KUKA KRL program: MyProgram_313().src

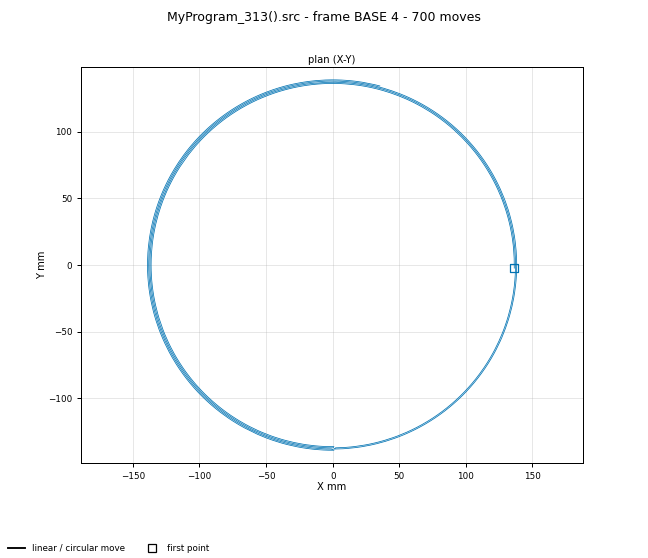
[picture p0: tool path of MyProgram_313().src in frame BASE 4, 700 of 700 moves have a stored position in this frame; points joined in program order, loops and branches not executed]
&ACCESS RVP
&REL 1
&PARAM TEMPLATE = C:\KRC\Roboter\Template\vorgabe
&PARAM EDITMASK = *
DEF MyProgram_313()
; ---- Setting reference (Base) ----
$BASE = BASE_DATA[4]

; --------------------------
; ---- Setting tool (TCP) ----
$TOOL = TOOL_DATA[3]
; --------------------------

$VEL.CP = VEL_APROX_PRINT
Startdeposition()
$VEL.CP = VEL_PRINT
LIN {X 136.3171,Y -2.3121,Z 183,A 1.901,B 4.2961,C 0.214,E1 4.4612,E2 450.9025} C_DIS
LIN {X 136.2426,Y 5.0697,Z 183,A 4.9757,B 4.2965,C 0.2056,E1 4.4611,E2 447.8295} C_DIS
LIN {X 135.7755,Y 12.3733,Z 183,A 8.1014,B 4.2969,C 0.1963,E1 4.4605,E2 444.6957} C_DIS
LIN {X 135.4586,Y 15.4613,Z 183,A 9.6734,B 4.2972,C 0.1892,E1 4.46,E2 443.0888} C_DIS
LIN {X 134.7828,Y 20.5264,Z 183,A 11.59,B 4.2974,C 0.1861,E1 4.4592,E2 441.2002} C_DIS
LIN {X 134.1353,Y 24.4028,Z 183,A 13.2335,B 4.2976,C 0.1816,E1 4.4584,E2 439.5567} C_DIS
LIN {X 133.2839,Y 28.6885,Z 183,A 14.8956,B 4.2976,C 0.1787,E1 4.4575,E2 437.9155} C_DIS
LIN {X 132.5463,Y 31.9229,Z 183,A 16.2711,B 4.2978,C 0.1751,E1 4.4566,E2 436.5415} C_DIS
LIN {X 131.506,Y 35.9772,Z 183,A 18.0412,B 4.298,C 0.1701,E1 4.4554,E2 434.7691} C_DIS
LIN {X 130.447,Y 39.6386,Z 183,A 19.5139,B 4.2981,C 0.1674,E1 4.4542,E2 433.3118} C_DIS
LIN {X 129.3994,Y 42.9345,Z 183,A 20.8992,B 4.2982,C 0.1643,E1 4.453,E2 431.9343} C_DIS
LIN {X 127.7702,Y 47.5649,Z 183,A 23.2775,B 4.2986,C 0.1549,E1 4.4507,E2 429.5151} C_DIS
LIN {X 126.4108,Y 51.0673,Z 183,A 24.4308,B 4.2986,C 0.156,E1 4.4496,E2 428.4147} C_DIS
LIN {X 125.0263,Y 54.3695,Z 183,A 25.8044,B 4.2986,C 0.1537,E1 4.4481,E2 427.0569} C_DIS
LIN {X 123.9979,Y 56.6781,Z 183,A 26.9937,B 4.2988,C 0.1494,E1 4.4467,E2 425.8511} C_DIS
LIN {X 122.4235,Y 60.0012,Z 183,A 28.472,B 4.2988,C 0.1462,E1 4.4449,E2 424.3805} C_DIS
LIN {X 120.7175,Y 63.3624,Z 183,A 29.8705,B 4.299,C 0.1445,E1 4.4431,E2 423.0045} C_DIS
LIN {X 118.9072,Y 66.7021,Z 183,A 31.598,B 4.2991,C 0.1389,E1 4.4408,E2 421.2601} C_DIS
LIN {X 116.1505,Y 71.3944,Z 183,A 33.7773,B 4.2993,C 0.1346,E1 4.4377,E2 419.0935} C_DIS
LIN {X 114.0434,Y 74.7147,Z 183,A 35.456,B 4.2994,C 0.1304,E1 4.4351,E2 417.411} C_DIS
LIN {X 111.5779,Y 78.3489,Z 183,A 37.2621,B 4.2995,C 0.1265,E1 4.4323,E2 415.6092} C_DIS
LIN {X 108.8614,Y 82.081,Z 183,A 38.9007,B 4.2995,C 0.1256,E1 4.4296,E2 414.0075} C_DIS
LIN {X 106.5784,Y 85.0244,Z 183,A 40.3825,B 4.2996,C 0.1231,E1 4.4271,E2 412.5356} C_DIS
LIN {X 103.9871,Y 88.1748,Z 183,A 42.3281,B 4.2998,C 0.1166,E1 4.4236,E2 410.5609} C_DIS
LIN {X 100.9585,Y 91.6267,Z 183,A 44.0964,B 4.2998,C 0.1144,E1 4.4203,E2 408.8123} C_DIS
LIN {X 96.8115,Y 95.9981,Z 183,A 46.6115,B 4.3,C 0.1093,E1 4.4155,E2 406.2989} C_DIS
LIN {X 91.1892,Y 101.3543,Z 183,A 49.8778,B 4.3002,C 0.1029,E1 4.4088,E2 403.0318} C_DIS
LIN {X 87.8086,Y 104.2966,Z 183,A 51.5269,B 4.3002,C 0.102,E1 4.4053,E2 401.4114} C_DIS
LIN {X 84.7834,Y 106.7702,Z 183,A 53.4489,B 4.3003,C 0.0958,E1 4.4011,E2 399.4547} C_DIS
LIN {X 80.5427,Y 110.0046,Z 183,A 55.502,B 4.3003,C 0.0941,E1 4.3965,E2 397.4248} C_DIS
LIN {X 76.9236,Y 112.5652,Z 183,A 57.3399,B 4.3004,C 0.0913,E1 4.3923,E2 395.5898} C_DIS
LIN {X 73.3431,Y 114.93,Z 183,A 59.0894,B 4.3004,C 0.089,E1 4.3882,E2 393.8469} C_DIS
LIN {X 69.468,Y 117.3134,Z 183,A 61.0062,B 4.3005,C 0.086,E1 4.3837,E2 391.9296} C_DIS
LIN {X 66.9374,Y 118.775,Z 183,A 62.2865,B 4.3005,C 0.0837,E1 4.3805,E2 390.6429} C_DIS
LIN {X 62.2571,Y 121.2921,Z 183,A 64.3036,B 4.3005,C 0.083,E1 4.3756,E2 388.6525} C_DIS
LIN {X 59.1852,Y 122.8204,Z 183,A 65.7141,B 4.3006,C 0.0814,E1 4.3721,E2 387.2459} C_DIS
LIN {X 55.8943,Y 124.352,Z 183,A 67.2309,B 4.3006,C 0.0796,E1 4.3682,E2 385.7304} C_DIS
LIN {X 52.4095,Y 125.8603,Z 183,A 68.781,B 4.3006,C 0.0782,E1 4.3643,E2 384.1861} C_DIS
LIN {X 49.7936,Y 126.9186,Z 183,A 69.9784,B 4.3006,C 0.0768,E1 4.3612,E2 382.9875} C_DIS
LIN {X 46.3245,Y 128.2248,Z 183,A 71.4966,B 4.3007,C 0.0756,E1 4.3572,E2 381.4743} C_DIS
LIN {X 43.3026,Y 129.2769,Z 183,A 72.8612,B 4.3007,C 0.0741,E1 4.3536,E2 380.1076} C_DIS
LIN {X 37.5599,Y 131.0627,Z 183,A 75.4609,B 4.3007,C 0.0711,E1 4.3466,E2 377.4997} C_DIS
LIN {X 33.8613,Y 132.0648,Z 183,A 76.9228,B 4.3007,C 0.0714,E1 4.3427,E2 376.0562} C_DIS
LIN {X 30.4313,Y 132.8967,Z 183,A 78.3894,B 4.3008,C 0.0705,E1 4.3387,E2 374.5921} C_DIS
LIN {X 27.0813,Y 133.6197,Z 183,A 79.8394,B 4.3008,C 0.0694,E1 4.3347,E2 373.1413} C_DIS
LIN {X 23.0702,Y 134.3719,Z 183,A 81.6264,B 4.3008,C 0.0678,E1 4.3298,E2 371.3461} C_DIS
LIN {X 19.4171,Y 134.9468,Z 183,A 83.0775,B 4.3008,C 0.068,E1 4.3258,E2 369.908} C_DIS
LIN {X 15.7292,Y 135.4268,Z 183,A 84.7916,B 4.3008,C 0.0659,E1 4.321,E2 368.1761} C_DIS
LIN {X 9.2863,Y 136.0215,Z 183,A 87.4726,B 4.3008,C 0.0654,E1 4.3136,E2 365.5008} C_DIS
LIN {X 6.3135,Y 136.1914,Z 183,A 89.0135,B 4.3009,C 0.0625,E1 4.3092,E2 363.925} C_DIS
LIN {X 2.4068,Y 136.3155,Z 183,A 90.1857,B 4.3009,C 0.0666,E1 4.3061,E2 362.811} C_DIS
LIN {X -4.4919,Y 136.2645,Z 183,A 93.2409,B 4.3009,C 0.0651,E1 4.2975,E2 359.7382} C_DIS
LIN {X -7.6288,Y 136.1251,Z 183,A 94.8342,B 4.3009,C 0.0628,E1 4.293,E2 358.1122} C_DIS
LIN {X -11.2331,Y 135.8732,Z 183,A 96.4152,B 4.3009,C 0.0624,E1 4.2885,E2 356.5241} C_DIS
LIN {X -15.4058,Y 135.4654,Z 183,A 97.8169,B 4.3009,C 0.0661,E1 4.2848,E2 355.1675} C_DIS
LIN {X -19.1221,Y 134.9889,Z 183,A 99.3275,B 4.3009,C 0.0671,E1 4.2806,E2 353.6654} C_DIS
LIN {X -22.8425,Y 134.4099,Z 183,A 100.9834,B 4.3009,C 0.0671,E1 4.276,E2 352.0014} C_DIS
LIN {X -26.9856,Y 133.6392,Z 183,A 102.6495,B 4.3009,C 0.0688,E1 4.2715,E2 350.3491} C_DIS
LIN {X -30.2949,Y 132.9279,Z 183,A 104.1186,B 4.3009,C 0.0692,E1 4.2674,E2 348.8751} C_DIS
LIN {X -33.6005,Y 132.131,Z 183,A 105.5284,B 4.3009,C 0.0703,E1 4.2636,E2 347.4684} C_DIS
LIN {X -36.8669,Y 131.2572,Z 183,A 107.3431,B 4.3009,C 0.0679,E1 4.2586,E2 345.6065} C_DIS
LIN {X -40.3293,Y 130.2356,Z 183,A 108.5381,B 4.3008,C 0.0718,E1 4.2555,E2 344.4519} C_DIS
LIN {X -44.2179,Y 128.9673,Z 183,A 110.2866,B 4.3008,C 0.073,E1 4.2509,E2 342.7009} C_DIS
LIN {X -47.9543,Y 127.6243,Z 183,A 112.7044,B 4.3008,C 0.0684,E1 4.2444,E2 340.1923} C_DIS
LIN {X -53.3534,Y 125.4656,Z 183,A 114.5344,B 4.3008,C 0.0759,E1 4.2398,E2 338.4394} C_DIS
LIN {X -56.6873,Y 123.9937,Z 183,A 115.9395,B 4.3007,C 0.0786,E1 4.2363,E2 337.0507} C_DIS
LIN {X -60.5692,Y 122.1433,Z 183,A 118.2237,B 4.3007,C 0.077,E1 4.2304,E2 334.7094} C_DIS
LIN {X -64.1356,Y 120.3106,Z 183,A 119.788,B 4.3007,C 0.0801,E1 4.2266,E2 333.1611} C_DIS
LIN {X -68.8121,Y 117.699,Z 183,A 121.7265,B 4.3005,C 0.0855,E1 4.222,E2 331.2625} C_DIS
LIN {X -72.0312,Y 115.7566,Z 183,A 123.5706,B 4.3005,C 0.0858,E1 4.2175,E2 329.3873} C_DIS
LIN {X -76.0435,Y 113.162,Z 183,A 125.5858,B 4.3005,C 0.0888,E1 4.2128,E2 327.3728} C_DIS
LIN {X -79.7494,Y 110.5813,Z 183,A 127.2851,B 4.3004,C 0.0933,E1 4.209,E2 325.6992} C_DIS
LIN {X -83.2352,Y 107.9819,Z 183,A 129.5008,B 4.3004,C 0.0935,E1 4.204,E2 323.4374} C_DIS
LIN {X -87.134,Y 104.8609,Z 183,A 131.4864,B 4.3003,C 0.098,E1 4.1997,E2 321.4673} C_DIS
LIN {X -90.591,Y 101.8896,Z 183,A 133.3086,B 4.3002,C 0.1021,E1 4.1959,E2 319.658} C_DIS
LIN {X -93.6569,Y 99.0781,Z 183,A 135.4627,B 4.3002,C 0.1026,E1 4.1914,E2 317.4555} C_DIS
LIN {X -96.0676,Y 96.7424,Z 183,A 136.6668,B 4.3001,C 0.1068,E1 4.189,E2 316.2779} C_DIS
LIN {X -99.1593,Y 93.5709,Z 183,A 138.5814,B 4.3,C 0.1102,E1 4.1853,E2 314.3582} C_DIS
LIN {X -103.3949,Y 88.8684,Z 183,A 141.4274,B 4.2999,C 0.1145,E1 4.18,E2 311.4916} C_DIS
LIN {X -108.2215,Y 82.9229,Z 183,A 144.6315,B 4.2997,C 0.1216,E1 4.1745,E2 308.2919} C_DIS
LIN {X -114.6392,Y 73.7974,Z 183,A 149.4868,B 4.2994,C 0.1314,E1 4.1668,E2 303.4203} C_DIS
LIN {X -117.1451,Y 69.7504,Z 183,A 151.5284,B 4.2992,C 0.136,E1 4.1638,E2 301.3752} C_DIS
LIN {X -119.4339,Y 65.7552,Z 183,A 153.5195,B 4.2991,C 0.1403,E1 4.161,E2 299.3788} C_DIS
LIN {X -121.3098,Y 62.2224,Z 183,A 155.1705,B 4.2989,C 0.1448,E1 4.1589,E2 297.7327} C_DIS
LIN {X -122.8831,Y 59.054,Z 183,A 156.4617,B 4.2988,C 0.1498,E1 4.1574,E2 296.467} C_DIS
LIN {X -124.4309,Y 55.7179,Z 183,A 158.7322,B 4.2988,C 0.1491,E1 4.1547,E2 294.1077} C_DIS
LIN {X -126.1198,Y 51.788,Z 183,A 160.2755,B 4.2986,C 0.1554,E1 4.153,E2 292.5978} C_DIS
LIN {X -127.6596,Y 47.8601,Z 183,A 161.7935,B 4.2983,C 0.1617,E1 4.1515,E2 291.1127} C_DIS
LIN {X -129.1595,Y 43.6552,Z 183,A 163.9661,B 4.2983,C 0.1649,E1 4.1495,E2 288.9049} C_DIS
LIN {X -131.0998,Y 37.4294,Z 183,A 166.8614,B 4.298,C 0.1713,E1 4.1472,E2 285.9926} C_DIS
LIN {X -132.0998,Y 33.7234,Z 183,A 168.3203,B 4.2978,C 0.1767,E1 4.1461,E2 284.5541} C_DIS
LIN {X -132.8008,Y 30.8514,Z 183,A 170.296,B 4.2978,C 0.1755,E1 4.1449,E2 282.4877} C_DIS
LIN {X -133.8259,Y 26.047,Z 183,A 171.8547,B 4.2974,C 0.1845,E1 4.144,E2 280.9941} C_DIS
LIN {X -134.4481,Y 22.6131,Z 183,A 173.3375,B 4.2973,C 0.1885,E1 4.1433,E2 279.5103} C_DIS
LIN {X -134.9784,Y 19.1958,Z 183,A 174.8432,B 4.2971,C 0.1922,E1 4.1427,E2 277.9992} C_DIS
LIN {X -135.4712,Y 15.3557,Z 183,A 176.5479,B 4.2969,C 0.1963,E1 4.1421,E2 276.2861} C_DIS
LIN {X -135.8304,Y 11.7403,Z 183,A 178.1035,B 4.2967,C 0.2004,E1 4.1417,E2 274.7279} C_DIS
LIN {X -136.0632,Y 8.6339,Z 183,A 179.5198,B 4.2966,C 0.2035,E1 4.1414,E2 273.2991} C_DIS
LIN {X -136.2696,Y 4.3069,Z 183,A -178.5717,B 4.2964,C 0.2081,E1 4.1412,E2 271.381} C_DIS
LIN {X -136.3402,Y 0.0169,Z 183,A -176.6762,B 4.2961,C 0.2126,E1 4.1412,E2 269.4752} C_DIS
LIN {X -136.2832,Y -3.8175,Z 183,A -175.1085,B 4.2959,C 0.2174,E1 4.1412,E2 267.914} C_DIS
LIN {X -136.1045,Y -7.9634,Z 183,A -173.3102,B 4.2957,C 0.222,E1 4.1415,E2 266.1101} C_DIS
LIN {X -135.852,Y -11.4845,Z 183,A -171.7908,B 4.2955,C 0.226,E1 4.1419,E2 264.5871} C_DIS
LIN {X -135.4498,Y -15.5365,Z 183,A -169.9324,B 4.2952,C 0.2298,E1 4.1424,E2 262.7113} C_DIS
LIN {X -134.9598,Y -19.3256,Z 183,A -168.3468,B 4.295,C 0.2345,E1 4.143,E2 261.1292} C_DIS
LIN {X -134.3387,Y -23.2663,Z 183,A -166.5398,B 4.2948,C 0.2383,E1 4.1439,E2 259.3068} C_DIS
LIN {X -133.6182,Y -27.0889,Z 183,A -164.9906,B 4.2945,C 0.2434,E1 4.1447,E2 257.7693} C_DIS
LIN {X -132.8825,Y -30.4937,Z 183,A -163.4974,B 4.2943,C 0.2472,E1 4.1456,E2 256.2733} C_DIS
LIN {X -131.3136,Y -36.6651,Z 183,A -160.6385,B 4.2939,C 0.2533,E1 4.1476,E2 253.3929} C_DIS
LIN {X -130.3246,Y -40.0388,Z 183,A -159.0904,B 4.2937,C 0.2568,E1 4.1489,E2 251.8366} C_DIS
LIN {X -127.4621,Y -48.3873,Z 183,A -155.2423,B 4.2932,C 0.2658,E1 4.1525,E2 247.9729} C_DIS
LIN {X -126.0166,Y -52.0351,Z 183,A -153.5708,B 4.2929,C 0.2699,E1 4.1542,E2 246.2993} C_DIS
LIN {X -124.6389,Y -55.253,Z 183,A -152.0835,B 4.2927,C 0.2736,E1 4.1559,E2 244.8106} C_DIS
LIN {X -123.2925,Y -58.197,Z 183,A -150.6015,B 4.2925,C 0.2762,E1 4.1576,E2 243.3138} C_DIS
LIN {X -121.615,Y -61.6229,Z 183,A -148.8042,B 4.2923,C 0.2789,E1 4.1599,E2 241.4922} C_DIS
LIN {X -119.1403,Y -66.2853,Z 183,A -146.405,B 4.2921,C 0.283,E1 4.1632,E2 239.0706} C_DIS
LIN {X -117.4157,Y -69.2945,Z 183,A -145.1492,B 4.2918,C 0.2879,E1 4.1649,E2 237.8414} C_DIS
LIN {X -115.0574,Y -73.1442,Z 183,A -143.1656,B 4.2915,C 0.2918,E1 4.1678,E2 235.8474} C_DIS
LIN {X -112.577,Y -76.9063,Z 183,A -141.2209,B 4.2912,C 0.2958,E1 4.1709,E2 233.8967} C_DIS
LIN {X -110.2635,Y -80.1879,Z 183,A -139.4641,B 4.291,C 0.2991,E1 4.1738,E2 232.1315} C_DIS
LIN {X -107.429,Y -83.9477,Z 183,A -137.4443,B 4.2907,C 0.3031,E1 4.1772,E2 230.107} C_DIS
LIN {X -104.6125,Y -87.4321,Z 183,A -135.5524,B 4.2904,C 0.307,E1 4.1806,E2 228.2145} C_DIS
LIN {X -102.418,Y -89.9933,Z 183,A -134.0693,B 4.2903,C 0.3095,E1 4.1833,E2 226.7231} C_DIS
LIN {X -98.7006,Y -94.0548,Z 183,A -131.7155,B 4.2899,C 0.3138,E1 4.1878,E2 224.3646} C_DIS
LIN {X -96.2337,Y -96.5774,Z 183,A -130.3834,B 4.2896,C 0.3178,E1 4.1904,E2 223.0524} C_DIS
LIN {X -93.7595,Y -98.9814,Z 183,A -128.7043,B 4.2896,C 0.3188,E1 4.1938,E2 221.3438} C_DIS
LIN {X -90.5069,Y -101.964,Z 183,A -126.8241,B 4.2893,C 0.3219,E1 4.1977,E2 219.4605} C_DIS
LIN {X -87.0847,Y -104.9017,Z 183,A -124.8812,B 4.2891,C 0.3248,E1 4.2019,E2 217.5117} C_DIS
LIN {X -83.4222,Y -107.837,Z 183,A -122.8734,B 4.2889,C 0.3278,E1 4.2063,E2 215.4994} C_DIS
LIN {X -79.771,Y -110.5656,Z 183,A -121.0017,B 4.2886,C 0.3312,E1 4.2105,E2 213.6335} C_DIS
LIN {X -76.2754,Y -113.0052,Z 183,A -119.1733,B 4.2884,C 0.3336,E1 4.2147,E2 211.8003} C_DIS
LIN {X -73.143,Y -115.0581,Z 183,A -117.4666,B 4.2884,C 0.3348,E1 4.2188,E2 210.0763} C_DIS
LIN {X -69.7634,Y -117.1373,Z 183,A -115.7098,B 4.2882,C 0.3363,E1 4.223,E2 208.3079} C_DIS
LIN {X -65.4726,Y -119.5888,Z 183,A -113.6904,B 4.288,C 0.3394,E1 4.2279,E2 206.2959} C_DIS
LIN {X -62.3781,Y -121.2305,Z 183,A -112.2243,B 4.2879,C 0.3412,E1 4.2316,E2 204.8304} C_DIS
LIN {X -59.177,Y -122.8243,Z 183,A -110.8983,B 4.2876,C 0.3444,E1 4.2348,E2 203.5273} C_DIS
LIN {X -56.3296,Y -124.1573,Z 183,A -109.3311,B 4.2876,C 0.3437,E1 4.2389,E2 201.9279} C_DIS
LIN {X -52.8989,Y -125.6559,Z 183,A -107.8264,B 4.2875,C 0.3459,E1 4.2427,E2 200.4319} C_DIS
LIN {X -49.409,Y -127.0681,Z 183,A -106.2591,B 4.2874,C 0.3475,E1 4.2468,E2 198.8662} C_DIS
LIN {X -46.4075,Y -128.1949,Z 183,A -104.9422,B 4.2872,C 0.3489,E1 4.2502,E2 197.553} C_DIS
LIN {X -43.471,Y -129.2208,Z 183,A -103.3323,B 4.2874,C 0.3472,E1 4.2546,E2 195.9033} C_DIS
LIN {X -38.5666,Y -130.768,Z 183,A -101.3944,B 4.2871,C 0.3507,E1 4.2597,E2 193.9941} C_DIS
LIN {X -35.4538,Y -131.6462,Z 183,A -100.0022,B 4.2871,C 0.3513,E1 4.2635,E2 192.5972} C_DIS
LIN {X -32.1264,Y -132.4973,Z 183,A -98.557,B 4.287,C 0.352,E1 4.2674,E2 191.1514} C_DIS
LIN {X -29.0028,Y -133.216,Z 183,A -97.186,B 4.287,C 0.3525,E1 4.2711,E2 189.7768} C_DIS
LIN {X -25.6001,Y -133.9114,Z 183,A -95.7519,B 4.2869,C 0.3533,E1 4.2751,E2 188.3456} C_DIS
LIN {X -22.6007,Y -134.4502,Z 183,A -94.5199,B 4.2868,C 0.3542,E1 4.2784,E2 187.1195} C_DIS
LIN {X -19.4079,Y -134.9481,Z 183,A -92.2688,B 4.2875,C 0.3461,E1 4.285,E2 184.7502} C_DIS
LIN {X -13.2742,Y -135.689,Z 183,A -90.5042,B 4.2868,C 0.3545,E1 4.2896,E2 183.0945} C_DIS
LIN {X -9.9023,Y -135.9765,Z 183,A -88.6028,B 4.2871,C 0.35,E1 4.2951,E2 181.1294} C_DIS
LIN {X -5.6395,Y -136.2204,Z 183,A -87.4752,B 4.2866,C 0.3565,E1 4.298,E2 180.0887} C_DIS
LIN {X 0.9463,Y -136.3293,Z 183,A -85.9047,B 4.2856,C 0.3681,E1 4.3021,E2 178.6724} C_DIS
Enddeposition()
LIN {X 0.9463,Y -136.3293,Z 183,A -85.9053,B 4.2856,C 0.3681,E1 4.3021,E2 178.6731} C_DIS
Startdeposition()
$VEL.CP = VEL_PRINT
LIN {X 0.2601,Y -137.2384,Z 183,A -85.4933,B 4.2391,C 0.3624,E1 4.2564,E2 178.217} C_DIS
LIN {X -3.5849,Y -137.1911,Z 183,A -86.9897,B 4.2391,C 0.3615,E1 4.2522,E2 179.6999} C_DIS
LIN {X -8.3049,Y -136.9862,Z 183,A -89.3069,B 4.2389,C 0.3648,E1 4.2456,E2 182.0629} C_DIS
LIN {X -11.9801,Y -136.7144,Z 183,A -90.5859,B 4.2391,C 0.3622,E1 4.2421,E2 183.3087} C_DIS
LIN {X -16.1912,Y -136.2791,Z 183,A -92.2802,B 4.2392,C 0.3612,E1 4.2375,E2 184.9941} C_DIS
LIN {X -19.279,Y -135.8767,Z 183,A -94.0043,B 4.2389,C 0.3648,E1 4.2325,E2 186.774} C_DIS
LIN {X -23.4354,Y -135.2238,Z 183,A -95.4492,B 4.2392,C 0.3613,E1 4.2287,E2 188.179} C_DIS
LIN {X -27.2424,Y -134.5064,Z 183,A -96.8991,B 4.2394,C 0.3591,E1 4.2247,E2 189.6075} C_DIS
LIN {X -29.9628,Y -133.928,Z 183,A -98.1591,B 4.2394,C 0.3595,E1 4.2213,E2 190.8808} C_DIS
LIN {X -33.7684,Y -133.018,Z 183,A -99.7549,B 4.2394,C 0.3583,E1 4.2169,E2 192.472} C_DIS
LIN {X -37.2233,Y -132.0931,Z 183,A -101.3123,B 4.2394,C 0.3579,E1 4.2127,E2 194.0382} C_DIS
LIN {X -40.8878,Y -131.007,Z 183,A -103.0788,B 4.2394,C 0.3583,E1 4.2079,E2 195.8275} C_DIS
LIN {X -44.5595,Y -129.8025,Z 183,A -104.3666,B 4.2398,C 0.3542,E1 4.2046,E2 197.0731} C_DIS
LIN {X -47.8395,Y -128.6295,Z 183,A -105.9965,B 4.2398,C 0.3545,E1 4.2003,E2 198.7263} C_DIS
LIN {X -51.2367,Y -127.314,Z 183,A -107.5208,B 4.2398,C 0.3532,E1 4.1963,E2 200.2512} C_DIS
LIN {X -54.5588,Y -125.9261,Z 183,A -109.0138,B 4.24,C 0.3516,E1 4.1925,E2 201.7431} C_DIS
LIN {X -57.4805,Y -124.6196,Z 183,A -110.3802,B 4.2401,C 0.3504,E1 4.189,E2 203.1137} C_DIS
LIN {X -60.5172,Y -123.1736,Z 183,A -111.8923,B 4.2401,C 0.3498,E1 4.1852,E2 204.6399} C_DIS
LIN {X -63.6638,Y -121.577,Z 183,A -113.298,B 4.2404,C 0.3475,E1 4.1817,E2 206.0369} C_DIS
LIN {X -67.4381,Y -119.5271,Z 183,A -115.1334,B 4.2405,C 0.3456,E1 4.1772,E2 207.8781} C_DIS
LIN {X -70.8525,Y -117.5353,Z 183,A -116.9033,B 4.2406,C 0.3443,E1 4.1729,E2 209.6635} C_DIS
LIN {X -74.5041,Y -115.2553,Z 183,A -118.7553,B 4.2408,C 0.3422,E1 4.1685,E2 211.5227} C_DIS
LIN {X -78.2554,Y -112.7418,Z 183,A -120.6384,B 4.241,C 0.3394,E1 4.1642,E2 213.4054} C_DIS
LIN {X -81.7759,Y -110.2149,Z 183,A -122.5092,B 4.2412,C 0.3371,E1 4.1599,E2 215.2841} C_DIS
LIN {X -85.3945,Y -107.4354,Z 183,A -124.3352,B 4.2415,C 0.3333,E1 4.1559,E2 217.0998} C_DIS
LIN {X -88.1603,Y -105.1776,Z 183,A -126.1692,B 4.2415,C 0.3333,E1 4.1519,E2 218.978} C_DIS
LIN {X -90.708,Y -102.9889,Z 183,A -127.3956,B 4.2418,C 0.3295,E1 4.1494,E2 220.1816} C_DIS
LIN {X -93.9609,Y -100.0301,Z 183,A -129.2727,B 4.242,C 0.3265,E1 4.1455,E2 222.0638} C_DIS
LIN {X -96.2069,Y -97.8716,Z 183,A -130.8148,B 4.242,C 0.3258,E1 4.1424,E2 223.6367} C_DIS
LIN {X -98.5717,Y -95.4892,Z 183,A -131.7436,B 4.2425,C 0.3196,E1 4.1407,E2 224.5043} C_DIS
LIN {X -103.5219,Y -90.099,Z 183,A -135.1526,B 4.2428,C 0.316,E1 4.1342,E2 227.9585} C_DIS
LIN {X -106.4573,Y -86.6113,Z 183,A -137.107,B 4.2431,C 0.3124,E1 4.1307,E2 229.919} C_DIS
LIN {X -109.4579,Y -82.7862,Z 183,A -139.5581,B 4.2431,C 0.3109,E1 4.1264,E2 232.4234} C_DIS
LIN {X -111.8993,Y -79.4564,Z 183,A -141.0153,B 4.2436,C 0.3052,E1 4.1241,E2 233.8461} C_DIS
LIN {X -114.5103,Y -75.644,Z 183,A -142.9558,B 4.2439,C 0.3008,E1 4.1211,E2 235.7873} C_DIS
LIN {X -116.8963,Y -71.9018,Z 183,A -144.8729,B 4.2442,C 0.2969,E1 4.1182,E2 237.712} C_DIS
LIN {X -119.3495,Y -67.7522,Z 183,A -146.9295,B 4.2445,C 0.2924,E1 4.1154,E2 239.7734} C_DIS
LIN {X -121.3088,Y -64.1746,Z 183,A -148.7116,B 4.2448,C 0.2887,E1 4.113,E2 241.5648} C_DIS
LIN {X -123.0576,Y -60.7523,Z 183,A -150.2133,B 4.2451,C 0.284,E1 4.1111,E2 243.0528} C_DIS
LIN {X -124.4866,Y -57.768,Z 183,A -151.7131,B 4.2453,C 0.2813,E1 4.1093,E2 244.5671} C_DIS
LIN {X -126.0422,Y -54.2902,Z 183,A -153.312,B 4.2455,C 0.2773,E1 4.1075,E2 246.1662} C_DIS
LIN {X -127.3248,Y -51.2098,Z 183,A -154.7888,B 4.2457,C 0.2742,E1 4.1059,E2 247.653} C_DIS
LIN {X -128.4892,Y -48.2141,Z 183,A -156.451,B 4.2458,C 0.2728,E1 4.1043,E2 249.3551} C_DIS
LIN {X -129.6279,Y -45.063,Z 183,A -157.6634,B 4.2461,C 0.2679,E1 4.1032,E2 250.5432} C_DIS
LIN {X -130.9576,Y -41.0455,Z 183,A -159.5558,B 4.2464,C 0.264,E1 4.1015,E2 252.4507} C_DIS
LIN {X -132.0714,Y -37.3007,Z 183,A -161.11,B 4.2467,C 0.2591,E1 4.1003,E2 253.9942} C_DIS
LIN {X -133.2683,Y -32.7729,Z 183,A -163.2089,B 4.2469,C 0.2547,E1 4.0989,E2 256.1102} C_DIS
LIN {X -134.101,Y -29.173,Z 183,A -164.7257,B 4.2472,C 0.2503,E1 4.0979,E2 257.6228} C_DIS
LIN {X -134.7767,Y -25.8722,Z 183,A -166.1765,B 4.2474,C 0.2466,E1 4.0971,E2 259.0783} C_DIS
LIN {X -135.4035,Y -22.3621,Z 183,A -167.7293,B 4.2476,C 0.2429,E1 4.0964,E2 260.6383} C_DIS
LIN {X -136.0284,Y -18.181,Z 183,A -169.5698,B 4.2479,C 0.2384,E1 4.0957,E2 262.4872} C_DIS
LIN {X -136.4568,Y -14.6181,Z 183,A -170.9903,B 4.2481,C 0.2337,E1 4.0952,E2 263.8969} C_DIS
LIN {X -136.7536,Y -11.5159,Z 183,A -172.396,B 4.2483,C 0.2307,E1 4.0949,E2 265.315} C_DIS
LIN {X -136.9966,Y -8.1356,Z 183,A -174.0188,B 4.2484,C 0.228,E1 4.0946,E2 266.9629} C_DIS
LIN {X -137.1858,Y -3.7744,Z 183,A -175.8124,B 4.2487,C 0.2227,E1 4.0944,E2 268.7516} C_DIS
LIN {X -137.2396,Y -0.3029,Z 183,A -177.4372,B 4.2489,C 0.2197,E1 4.0944,E2 270.3974} C_DIS
LIN {X -137.1862,Y 3.7592,Z 183,A -179.0703,B 4.2491,C 0.2145,E1 4.0944,E2 272.0214} C_DIS
LIN {X -137.0072,Y 7.9645,Z 183,A 179.0956,B 4.2494,C 0.21,E1 4.0947,E2 273.8638} C_DIS
LIN {X -136.7496,Y 11.5627,Z 183,A 177.5779,B 4.2496,C 0.2058,E1 4.095,E2 275.3819} C_DIS
LIN {X -136.368,Y 15.4439,Z 183,A 175.7995,B 4.2498,C 0.2021,E1 4.0956,E2 277.1778} C_DIS
LIN {X -135.8787,Y 19.2647,Z 183,A 174.1963,B 4.25,C 0.1976,E1 4.0962,E2 278.7791} C_DIS
LIN {X -135.2411,Y 23.3353,Z 183,A 172.3171,B 4.2501,C 0.1937,E1 4.097,E2 280.6768} C_DIS
LIN {X -134.5025,Y 27.2619,Z 183,A 170.6317,B 4.2503,C 0.1892,E1 4.0979,E2 282.363} C_DIS
LIN {X -133.5396,Y 31.6473,Z 183,A 168.6557,B 4.2505,C 0.1847,E1 4.0992,E2 284.3502} C_DIS
LIN {X -132.5441,Y 35.5839,Z 183,A 166.9366,B 4.2507,C 0.1802,E1 4.1004,E2 286.0709} C_DIS
LIN {X -131.6299,Y 38.8295,Z 183,A 165.4351,B 4.2509,C 0.1769,E1 4.1016,E2 287.5829} C_DIS
LIN {X -130.3284,Y 42.9967,Z 183,A 163.606,B 4.2511,C 0.172,E1 4.1031,E2 289.4113} C_DIS
LIN {X -128.9393,Y 46.9993,Z 183,A 161.7571,B 4.2512,C 0.1678,E1 4.1049,E2 291.2687} C_DIS
LIN {X -127.6226,Y 50.4694,Z 183,A 160.2723,B 4.2514,C 0.1633,E1 4.1063,E2 292.7443} C_DIS
LIN {X -124.1756,Y 58.4387,Z 183,A 156.4308,B 4.2517,C 0.1553,E1 4.1107,E2 296.6097} C_DIS
LIN {X -122.4671,Y 61.9351,Z 183,A 154.8796,B 4.2519,C 0.1507,E1 4.1126,E2 298.1504} C_DIS
LIN {X -120.7035,Y 65.3101,Z 183,A 153.1135,B 4.2519,C 0.1479,E1 4.115,E2 299.937} C_DIS
LIN {X -118.5431,Y 69.1542,Z 183,A 151.1725,B 4.2521,C 0.144,E1 4.1177,E2 301.8887} C_DIS
LIN {X -116.1965,Y 73.0276,Z 183,A 149.3029,B 4.2523,C 0.1394,E1 4.1204,E2 303.7542} C_DIS
LIN {X -112.8084,Y 78.1596,Z 183,A 146.6334,B 4.2524,C 0.134,E1 4.1246,E2 306.4341} C_DIS
LIN {X -110.3698,Y 81.5674,Z 183,A 144.8068,B 4.2525,C 0.1306,E1 4.1276,E2 308.2687} C_DIS
LIN {X -107.6211,Y 85.1612,Z 183,A 142.8691,B 4.2527,C 0.1267,E1 4.1309,E2 310.2108} C_DIS
LIN {X -105.2665,Y 88.0544,Z 183,A 141.1005,B 4.2527,C 0.1248,E1 4.1341,E2 312.0039} C_DIS
LIN {X -101.563,Y 92.3014,Z 183,A 138.8869,B 4.2529,C 0.1189,E1 4.1382,E2 314.1987} C_DIS
LIN {X -98.5484,Y 95.5133,Z 183,A 137.0517,B 4.2529,C 0.1152,E1 4.1417,E2 316.032} C_DIS
LIN {X -95.8654,Y 98.2064,Z 183,A 135.4977,B 4.2531,C 0.1118,E1 4.1448,E2 317.5807} C_DIS
LIN {X -93.7361,Y 100.2407,Z 183,A 134.0774,B 4.2531,C 0.1108,E1 4.1477,E2 319.0232} C_DIS
LIN {X -90.3316,Y 103.3189,Z 183,A 132.1482,B 4.2531,C 0.1073,E1 4.1517,E2 320.9525} C_DIS
LIN {X -87.1051,Y 106.0538,Z 183,A 130.3098,B 4.2533,C 0.1047,E1 4.1557,E2 322.7983} C_DIS
LIN {X -84.2489,Y 108.3363,Z 183,A 128.9662,B 4.2533,C 0.1008,E1 4.1586,E2 324.1185} C_DIS
LIN {X -81.3703,Y 110.5146,Z 183,A 127.2372,B 4.2533,C 0.0999,E1 4.1625,E2 325.8734} C_DIS
LIN {X -77.6878,Y 113.1335,Z 183,A 125.3605,B 4.2534,C 0.0969,E1 4.1668,E2 327.7475} C_DIS
LIN {X -74.1226,Y 115.5009,Z 183,A 123.5147,B 4.2534,C 0.0946,E1 4.1711,E2 329.5991} C_DIS
LIN {X -71.0384,Y 117.4229,Z 183,A 121.7051,B 4.2534,C 0.0946,E1 4.1756,E2 331.4429} C_DIS
LIN {X -67.9666,Y 119.2272,Z 183,A 120.4764,B 4.2536,C 0.0907,E1 4.1784,E2 332.6394} C_DIS
LIN {X -65.2687,Y 120.7257,Z 183,A 118.4359,B 4.2535,C 0.0947,E1 4.1837,E2 334.7696} C_DIS
LIN {X -60.0003,Y 123.4286,Z 183,A 116.5624,B 4.2537,C 0.0872,E1 4.1882,E2 336.5694} C_DIS
LIN {X -56.4517,Y 125.0897,Z 183,A 115.0754,B 4.2537,C 0.0842,E1 4.1919,E2 338.0373} C_DIS
LIN {X -53.1906,Y 126.5105,Z 183,A 113.2957,B 4.2537,C 0.0849,E1 4.1966,E2 339.8516} C_DIS
LIN {X -49.0237,Y 128.1846,Z 183,A 111.5771,B 4.2537,C 0.0819,E1 4.201,E2 341.5501} C_DIS
LIN {X -45.4743,Y 129.4853,Z 183,A 110.0136,B 4.2537,C 0.0803,E1 4.2051,E2 343.1108} C_DIS
LIN {X -41.9569,Y 130.6665,Z 183,A 108.5035,B 4.2538,C 0.0787,E1 4.2091,E2 344.6152} C_DIS
LIN {X -39.0993,Y 131.5509,Z 183,A 107.3572,B 4.2538,C 0.077,E1 4.2121,E2 345.7484} C_DIS
LIN {X -35.6948,Y 132.5145,Z 183,A 105.7334,B 4.2538,C 0.0772,E1 4.2166,E2 347.3891} C_DIS
LIN {X -32.4552,Y 133.3448,Z 183,A 104.4011,B 4.2538,C 0.0758,E1 4.2201,E2 348.7128} C_DIS
LIN {X -29.1429,Y 134.1075,Z 183,A 103.0262,B 4.2538,C 0.0746,E1 4.2239,E2 350.0815} C_DIS
LIN {X -26.5653,Y 134.6442,Z 183,A 101.7012,B 4.2538,C 0.076,E1 4.2276,E2 351.4333} C_DIS
LIN {X -23.1425,Y 135.2733,Z 183,A 100.2784,B 4.2538,C 0.0751,E1 4.2315,E2 352.8516} C_DIS
LIN {X -19.2564,Y 135.8799,Z 183,A 98.6936,B 4.2539,C 0.074,E1 4.2358,E2 354.4286} C_DIS
LIN {X -15.59,Y 136.3508,Z 183,A 97.2032,B 4.2539,C 0.0732,E1 4.24,E2 355.9119} C_DIS
LIN {X -5.2554,Y 137.137,Z 183,A 92.7993,B 4.2539,C 0.0733,E1 4.2523,E2 360.3231} C_DIS
LIN {X 2.0919,Y 137.2219,Z 183,A 89.9384,B 4.2539,C 0.0716,E1 4.2602,E2 363.1577} C_DIS
LIN {X 9.3172,Y 136.9227,Z 183,A 85.9601,B 4.2538,C 0.0811,E1 4.2716,E2 367.2506} C_DIS
LIN {X 15.2036,Y 136.3938,Z 183,A 83.8558,B 4.2538,C 0.0787,E1 4.2773,E2 369.3105} C_DIS
LIN {X 19.1599,Y 135.8937,Z 183,A 82.6308,B 4.2538,C 0.0752,E1 4.2806,E2 370.4817} C_DIS
LIN {X 22.5717,Y 135.3685,Z 183,A 81.2103,B 4.2538,C 0.0758,E1 4.2845,E2 371.8993} C_DIS
LIN {X 26.2511,Y 134.7043,Z 183,A 79.6483,B 4.2538,C 0.0767,E1 4.2888,E2 373.4609} C_DIS
LIN {X 30.1207,Y 133.8919,Z 183,A 77.9549,B 4.2538,C 0.0782,E1 4.2934,E2 375.1591} C_DIS
LIN {X 33.7685,Y 133.018,Z 183,A 76.4358,B 4.2538,C 0.0789,E1 4.2975,E2 376.672} C_DIS
LIN {X 37.1198,Y 132.122,Z 183,A 75.0255,B 4.2538,C 0.0797,E1 4.3013,E2 378.0774} C_DIS
LIN {X 40.6062,Y 131.0932,Z 183,A 73.4777,B 4.2538,C 0.0814,E1 4.3054,E2 379.6285} C_DIS
LIN {X 44.7566,Y 129.7341,Z 183,A 71.7204,B 4.2538,C 0.0825,E1 4.3101,E2 381.3775} C_DIS
LIN {X 48.1002,Y 128.5318,Z 183,A 70.3349,B 4.2538,C 0.083,E1 4.3137,E2 382.7508} C_DIS
LIN {X 50.9035,Y 127.4483,Z 183,A 69.0172,B 4.2537,C 0.085,E1 4.3171,E2 384.076} C_DIS
LIN {X 54.1583,Y 126.0993,Z 183,A 67.5527,B 4.2537,C 0.0867,E1 4.3209,E2 385.5395} C_DIS
LIN {X 56.8125,Y 124.9283,Z 183,A 66.2204,B 4.2537,C 0.0894,E1 4.3243,E2 386.8864} C_DIS
LIN {X 60.3939,Y 123.2344,Z 183,A 64.6928,B 4.2536,C 0.0902,E1 4.3281,E2 388.3984} C_DIS
LIN {X 63.3851,Y 121.7233,Z 183,A 63.3232,B 4.2536,C 0.0918,E1 4.3315,E2 389.7644} C_DIS
LIN {X 67.3168,Y 119.5953,Z 183,A 61.4515,B 4.2535,C 0.0945,E1 4.3361,E2 391.6367} C_DIS
LIN {X 71.1732,Y 117.3414,Z 183,A 59.6076,B 4.2535,C 0.0971,E1 4.3405,E2 393.478} C_DIS
LIN {X 74.9729,Y 114.951,Z 183,A 57.7763,B 4.2534,C 0.0996,E1 4.3448,E2 395.3041} C_DIS
LIN {X 78.6365,Y 112.4766,Z 183,A 55.9552,B 4.2534,C 0.1023,E1 4.349,E2 397.1222} C_DIS
LIN {X 82.3156,Y 109.8131,Z 183,A 54.124,B 4.2533,C 0.1049,E1 4.3531,E2 398.9456} C_DIS
LIN {X 85.1425,Y 107.636,Z 183,A 52.6724,B 4.2533,C 0.1071,E1 4.3563,E2 400.3926} C_DIS
LIN {X 88.4415,Y 104.9418,Z 183,A 50.8999,B 4.2531,C 0.1103,E1 4.3601,E2 402.1646} C_DIS
LIN {X 91.8238,Y 101.9955,Z 183,A 49.2461,B 4.2531,C 0.1114,E1 4.3635,E2 403.7917} C_DIS
LIN {X 95.0082,Y 99.0358,Z 183,A 47.3155,B 4.253,C 0.1163,E1 4.3675,E2 405.7369} C_DIS
LIN {X 98.0163,Y 96.0593,Z 183,A 45.5879,B 4.2529,C 0.1195,E1 4.3709,E2 407.4599} C_DIS
LIN {X 101.4659,Y 92.4085,Z 183,A 43.5176,B 4.2528,C 0.1236,E1 4.3748,E2 409.5274} C_DIS
LIN {X 104.3986,Y 89.0819,Z 183,A 41.9021,B 4.2528,C 0.1249,E1 4.3777,E2 411.1142} C_DIS
LIN {X 106.6747,Y 86.3432,Z 183,A 40.2547,B 4.2526,C 0.13,E1 4.3807,E2 412.7819} C_DIS
LIN {X 109.498,Y 82.7331,Z 183,A 38.4167,B 4.2525,C 0.1335,E1 4.3838,E2 414.6111} C_DIS
LIN {X 112.1777,Y 79.0617,Z 183,A 36.583,B 4.2523,C 0.1371,E1 4.3868,E2 416.4375} C_DIS
LIN {X 114.6261,Y 75.4681,Z 183,A 34.7176,B 4.2522,C 0.142,E1 4.3897,E2 418.3097} C_DIS
LIN {X 116.7641,Y 72.1168,Z 183,A 32.494,B 4.2518,C 0.1527,E1 4.3931,E2 420.6033} C_DIS
LIN {X 119.8418,Y 66.8783,Z 183,A 30.6879,B 4.2518,C 0.1503,E1 4.3954,E2 422.3204} C_DIS
LIN {X 122.0424,Y 62.7693,Z 183,A 28.9595,B 4.2518,C 0.1526,E1 4.3976,E2 424.0225} C_DIS
LIN {X 123.6104,Y 59.6218,Z 183,A 27.4164,B 4.2516,C 0.1572,E1 4.3995,E2 425.5756} C_DIS
LIN {X 124.8644,Y 56.9507,Z 183,A 25.9668,B 4.2514,C 0.163,E1 4.4012,E2 427.0528} C_DIS
LIN {X 126.3311,Y 53.6202,Z 183,A 24.8527,B 4.2514,C 0.1621,E1 4.4024,E2 428.1172} C_DIS
LIN {X 129.5505,Y 45.2862,Z 183,A 21.1951,B 4.2511,C 0.1711,E1 4.4061,E2 431.7678} C_DIS
LIN {X 130.6832,Y 41.9044,Z 183,A 19.7829,B 4.251,C 0.1742,E1 4.4073,E2 433.1711} C_DIS
LIN {X 131.5455,Y 39.1177,Z 183,A 18.6917,B 4.251,C 0.1759,E1 4.4081,E2 434.2471} C_DIS
LIN {X 132.522,Y 35.6666,Z 183,A 17.1592,B 4.2507,C 0.1804,E1 4.4093,E2 435.7849} C_DIS
LIN {X 133.3338,Y 32.501,Z 183,A 15.7812,B 4.2506,C 0.1844,E1 4.4102,E2 437.1653} C_DIS
LIN {X 134.1767,Y 28.8227,Z 183,A 14.2727,B 4.2504,C 0.1879,E1 4.4111,E2 438.6663} C_DIS
LIN {X 134.9959,Y 24.7086,Z 183,A 12.5496,B 4.2502,C 0.1924,E1 4.412,E2 440.387} C_DIS
LIN {X 135.6149,Y 21.0411,Z 183,A 11.14,B 4.2501,C 0.195,E1 4.4126,E2 441.7795} C_DIS
LIN {X 136.6279,Y 12.9236,Z 183,A 8.0397,B 4.2498,C 0.2007,E1 4.4137,E2 444.8422} C_DIS
LIN {X 137.095,Y 6.2856,Z 183,A 5.012,B 4.2493,C 0.2117,E1 4.4143,E2 447.9035} C_DIS
LIN {X 137.2248,Y 1.9179,Z 183,A 3.5215,B 4.2493,C 0.2126,E1 4.4143,E2 449.3529} C_DIS
LIN {X 137.2147,Y -2.523,Z 183,A 0.9632,B 4.2485,C 0.2267,E1 4.4143,E2 452.0017} C_DIS
LIN {X 137.0297,Y -7.5842,Z 183,A -0.6182,B 4.2485,C 0.226,E1 4.414,E2 453.5174} C_DIS
LIN {X 136.7543,Y -11.507,Z 183,A -2.0858,B 4.2485,C 0.2285,E1 4.4137,E2 454.964} C_DIS
LIN {X 136.3268,Y -15.7918,Z 183,A -4.3515,B 4.2478,C 0.2394,E1 4.413,E2 457.2905} C_DIS
LIN {X 135.7093,Y -20.4313,Z 183,A -5.799,B 4.2478,C 0.2386,E1 4.4125,E2 458.6752} C_DIS
LIN {X 135.1052,Y -24.0976,Z 183,A -7.2061,B 4.2478,C 0.2411,E1 4.4118,E2 460.0651} C_DIS
LIN {X 134.4141,Y -27.6961,Z 183,A -8.7194,B 4.2475,C 0.2452,E1 4.411,E2 461.5775} C_DIS
LIN {X 133.4871,Y -31.865,Z 183,A -10.3454,B 4.2473,C 0.2482,E1 4.41,E2 463.1848} C_DIS
LIN {X 132.6589,Y -35.1532,Z 183,A -11.7898,B 4.2471,C 0.2524,E1 4.409,E2 464.634} C_DIS
LIN {X 131.811,Y -38.211,Z 183,A -13.1026,B 4.2469,C 0.2559,E1 4.408,E2 465.9464} C_DIS
LIN {X 130.8704,Y -41.3184,Z 183,A -14.2498,B 4.2468,C 0.257,E1 4.4071,E2 467.0679} C_DIS
LIN {X 129.7641,Y -44.6702,Z 183,A -15.6912,B 4.2466,C 0.2606,E1 4.4058,E2 468.5064} C_DIS
LIN {X 128.6314,Y -47.8342,Z 183,A -17.1793,B 4.2463,C 0.2654,E1 4.4044,E2 470.0066} C_DIS
LIN {X 127.3907,Y -51.0464,Z 183,A -18.545,B 4.2461,C 0.2684,E1 4.403,E2 471.3643} C_DIS
LIN {X 126.0619,Y -54.2449,Z 183,A -19.8367,B 4.246,C 0.2703,E1 4.4016,E2 472.6373} C_DIS
LIN {X 124.7503,Y -57.1979,Z 183,A -21.3296,B 4.2456,C 0.2756,E1 4.3999,E2 474.1499} C_DIS
LIN {X 123.2069,Y -60.4497,Z 183,A -22.7236,B 4.2455,C 0.2781,E1 4.3982,E2 475.5311} C_DIS
LIN {X 121.7286,Y -63.3751,Z 183,A -24.1103,B 4.2452,C 0.2818,E1 4.3964,E2 476.9214} C_DIS
LIN {X 120.4155,Y -65.8385,Z 183,A -25.6562,B 4.2447,C 0.2895,E1 4.3943,E2 478.5172} C_DIS
LIN {X 118.3071,Y -69.5559,Z 183,A -26.993,B 4.2447,C 0.2884,E1 4.3925,E2 479.7981} C_DIS
LIN {X 115.9705,Y -73.3857,Z 183,A -28.8103,B 4.2445,C 0.2923,E1 4.3898,E2 481.6098} C_DIS
LIN {X 113.6073,Y -76.9932,Z 183,A -30.6712,B 4.2442,C 0.2974,E1 4.3869,E2 483.48} C_DIS
LIN {X 110.3992,Y -81.5274,Z 183,A -32.8528,B 4.2439,C 0.3012,E1 4.3834,E2 485.6458} C_DIS
LIN {X 107.6807,Y -85.0858,Z 183,A -34.6919,B 4.2436,C 0.3051,E1 4.3802,E2 487.4826} C_DIS
LIN {X 104.8614,Y -88.5373,Z 183,A -36.4916,B 4.2434,C 0.3086,E1 4.377,E2 489.276} C_DIS
LIN {X 101.9666,Y -91.8561,Z 183,A -38.2829,B 4.2431,C 0.312,E1 4.3737,E2 491.0626} C_DIS
LIN {X 98.8913,Y -95.1592,Z 183,A -40.1362,B 4.2428,C 0.3157,E1 4.3701,E2 492.9135} C_DIS
LIN {X 95.695,Y -98.3726,Z 183,A -41.9875,B 4.2426,C 0.3191,E1 4.3665,E2 494.7611} C_DIS
LIN {X 92.3803,Y -101.4914,Z 183,A -43.8263,B 4.2424,C 0.3222,E1 4.3627,E2 496.5936} C_DIS
LIN {X 89.0094,Y -104.4602,Z 183,A -45.6571,B 4.2421,C 0.3253,E1 4.3589,E2 498.4201} C_DIS
LIN {X 85.3709,Y -107.4542,Z 183,A -47.5151,B 4.2419,C 0.3277,E1 4.3549,E2 500.2655} C_DIS
LIN {X 82.047,Y -110.0131,Z 183,A -49.2766,B 4.2417,C 0.331,E1 4.3509,E2 502.0297} C_DIS
LIN {X 78.4911,Y -112.5778,Z 183,A -51.0774,B 4.2415,C 0.3338,E1 4.3468,E2 503.8281} C_DIS
LIN {X 74.8544,Y -115.0279,Z 183,A -52.853,B 4.2413,C 0.3362,E1 4.3427,E2 505.5979} C_DIS
LIN {X 71.5264,Y -117.1266,Z 183,A -54.6288,B 4.2409,C 0.3404,E1 4.3385,E2 507.3924} C_DIS
LIN {X 67.0023,Y -119.7721,Z 183,A -56.6403,B 4.2409,C 0.3417,E1 4.3336,E2 509.3826} C_DIS
LIN {X 63.0307,Y -121.9093,Z 183,A -58.55,B 4.2406,C 0.3447,E1 4.3289,E2 511.2972} C_DIS
LIN {X 59.4257,Y -123.7041,Z 183,A -60.1042,B 4.2406,C 0.3455,E1 4.325,E2 512.8359} C_DIS
LIN {X 55.3459,Y -125.5844,Z 183,A -62.0285,B 4.2403,C 0.3485,E1 4.3201,E2 514.768} C_DIS
LIN {X 51.5704,Y -127.1795,Z 183,A -63.4715,B 4.2403,C 0.3476,E1 4.3165,E2 516.1771} C_DIS
LIN {X 48.9897,Y -128.1978,Z 183,A -64.8443,B 4.24,C 0.3513,E1 4.3128,E2 517.5788} C_DIS
LIN {X 45.4726,Y -129.4859,Z 183,A -66.3514,B 4.24,C 0.3523,E1 4.3089,E2 519.0796} C_DIS
LIN {X 41.9128,Y -130.6806,Z 183,A -67.8097,B 4.24,C 0.3527,E1 4.305,E2 520.5247} C_DIS
LIN {X 39.1474,Y -131.5368,Z 183,A -69.0868,B 4.2398,C 0.3546,E1 4.3016,E2 521.8116} C_DIS
LIN {X 35.2338,Y -132.6374,Z 183,A -70.7024,B 4.2398,C 0.3552,E1 4.2973,E2 523.4175} C_DIS
LIN {X 31.521,Y -133.57,Z 183,A -72.4032,B 4.2395,C 0.3576,E1 4.2926,E2 525.1327} C_DIS
LIN {X 27.2765,Y -134.4995,Z 183,A -73.9902,B 4.2396,C 0.3565,E1 4.2884,E2 526.6912} C_DIS
LIN {X 23.9799,Y -135.1263,Z 183,A -75.3629,B 4.2396,C 0.3571,E1 4.2846,E2 528.061} C_DIS
LIN {X 16.7639,Y -136.2108,Z 183,A -78.3613,B 4.2395,C 0.3583,E1 4.2763,E2 531.055} C_DIS
LIN {X 13.8693,Y -136.5368,Z 183,A -80.2655,B 4.2388,C 0.3658,E1 4.2708,E2 533.0496} C_DIS
LIN {X 9.0948,Y -136.9375,Z 183,A -81.875,B 4.2391,C 0.3626,E1 4.2664,E2 534.6094} C_DIS
LIN {X 2.1751,Y -137.2205,Z 183,A -84.5869,B 4.2391,C 0.3615,E1 4.2589,E2 537.2992} C_DIS
LIN {X 2.1751,Y -137.2205,Z 183,A -84.5869,B 4.2391,C 0.3615,E1 4.2589,E2 537.2992} C_DIS
Enddeposition()
LIN {X 0.9654,Y -138.1342,Z 183,A -84.4639,B 4.1943,C 0.3565,E1 4.2142,E2 537.138} C_DIS
Startdeposition()
$VEL.CP = VEL_PRINT
LIN {X 4.6091,Y -138.064,Z 183,A -82.7597,B 4.1945,C 0.3543,E1 4.219,E2 535.4075} C_DIS
LIN {X 7.7136,Y -137.9253,Z 183,A -81.6263,B 4.1944,C 0.3555,E1 4.2221,E2 534.2942} C_DIS
LIN {X 10.841,Y -137.7148,Z 183,A -80.1733,B 4.1946,C 0.3535,E1 4.2262,E2 532.8201} C_DIS
LIN {X 14.6117,Y -137.3637,Z 183,A -78.8026,B 4.1944,C 0.3548,E1 4.23,E2 531.4751} C_DIS
LIN {X 17.7428,Y -136.9945,Z 183,A -77.4604,B 4.1945,C 0.3539,E1 4.2337,E2 530.1277} C_DIS
LIN {X 21.9347,Y -136.3883,Z 183,A -75.713,B 4.1946,C 0.353,E1 4.2385,E2 528.3805} C_DIS
LIN {X 25.1365,Y -135.8347,Z 183,A -74.3735,B 4.1946,C 0.3522,E1 4.2422,E2 527.0413} C_DIS
LIN {X 28.3479,Y -135.201,Z 183,A -72.8832,B 4.1949,C 0.3499,E1 4.2463,E2 525.5325} C_DIS
LIN {X 33.1766,Y -134.0978,Z 183,A -70.9865,B 4.1949,C 0.3499,E1 4.2514,E2 523.6557} C_DIS
LIN {X 36.3993,Y -133.2591,Z 183,A -69.6175,B 4.1949,C 0.3489,E1 4.2551,E2 522.2873} C_DIS
LIN {X 39.6214,Y -132.3369,Z 183,A -68.1461,B 4.1951,C 0.3467,E1 4.2591,E2 520.8042} C_DIS
LIN {X 43.1404,Y -131.2302,Z 183,A -66.8414,B 4.1951,C 0.3476,E1 4.2625,E2 519.5285} C_DIS
LIN {X 46.1908,Y -130.1886,Z 183,A -65.4587,B 4.1952,C 0.3457,E1 4.2662,E2 518.1388} C_DIS
LIN {X 49.2529,Y -129.0622,Z 183,A -64.0683,B 4.1954,C 0.3438,E1 4.2698,E2 516.7425} C_DIS
LIN {X 52.4412,Y -127.7999,Z 183,A -62.5388,B 4.1956,C 0.3409,E1 4.2738,E2 515.1978} C_DIS
LIN {X 55.6128,Y -126.452,Z 183,A -61.2544,B 4.1956,C 0.3408,E1 4.2771,E2 513.9317} C_DIS
LIN {X 58.7645,Y -125.0185,Z 183,A -59.8392,B 4.1957,C 0.3391,E1 4.2807,E2 512.5182} C_DIS
LIN {X 61.8929,Y -123.4997,Z 183,A -58.4188,B 4.1959,C 0.3374,E1 4.2842,E2 511.0997} C_DIS
LIN {X 65.626,Y -121.5567,Z 183,A -56.6837,B 4.1961,C 0.335,E1 4.2885,E2 509.3646} C_DIS
LIN {X 69.3089,Y -119.4948,Z 183,A -54.9378,B 4.1963,C 0.3324,E1 4.2927,E2 507.618} C_DIS
LIN {X 72.8869,Y -117.3466,Z 183,A -53.1948,B 4.1965,C 0.3295,E1 4.2969,E2 505.8721} C_DIS
LIN {X 76.7802,Y -114.8369,Z 183,A -51.3496,B 4.1967,C 0.3272,E1 4.3012,E2 504.0355} C_DIS
LIN {X 80.4411,Y -112.3029,Z 183,A -49.5427,B 4.1969,C 0.3245,E1 4.3053,E2 502.2324} C_DIS
LIN {X 83.9131,Y -109.7329,Z 183,A -47.7656,B 4.1971,C 0.3215,E1 4.3093,E2 500.4558} C_DIS
LIN {X 87.5191,Y -106.879,Z 183,A -45.9247,B 4.1973,C 0.3187,E1 4.3133,E2 498.6222} C_DIS
LIN {X 90.7363,Y -104.1616,Z 183,A -44.1709,B 4.1976,C 0.3152,E1 4.317,E2 496.866} C_DIS
LIN {X 94.2213,Y -101.0201,Z 183,A -42.2884,B 4.1978,C 0.3121,E1 4.3209,E2 494.9904} C_DIS
LIN {X 97.4806,Y -97.8788,Z 183,A -40.489,B 4.1981,C 0.3092,E1 4.3244,E2 493.1997} C_DIS
LIN {X 100.5628,Y -94.7092,Z 183,A -38.6931,B 4.1983,C 0.3058,E1 4.3279,E2 491.4073} C_DIS
LIN {X 103.5728,Y -91.4078,Z 183,A -36.8875,B 4.1986,C 0.3023,E1 4.3313,E2 489.6064} C_DIS
LIN {X 106.4788,Y -88.0056,Z 183,A -35.0824,B 4.1988,C 0.2988,E1 4.3345,E2 487.8065} C_DIS
LIN {X 109.2551,Y -84.5343,Z 183,A -33.287,B 4.1991,C 0.2951,E1 4.3376,E2 486.0159} C_DIS
LIN {X 111.7834,Y -81.1616,Z 183,A -31.5444,B 4.1993,C 0.2911,E1 4.3405,E2 484.2726} C_DIS
LIN {X 114.4617,Y -77.3385,Z 183,A -29.7061,B 4.1996,C 0.2877,E1 4.3434,E2 482.4455} C_DIS
LIN {X 116.8538,Y -73.6743,Z 183,A -27.936,B 4.1998,C 0.2839,E1 4.346,E2 480.6798} C_DIS
LIN {X 119.0511,Y -70.0682,Z 183,A -26.202,B 4.2001,C 0.2797,E1 4.3485,E2 478.9467} C_DIS
LIN {X 121.2172,Y -66.2505,Z 183,A -24.6002,B 4.2002,C 0.2779,E1 4.3507,E2 477.3721} C_DIS
LIN {X 122.7083,Y -63.4474,Z 183,A -23.244,B 4.2005,C 0.274,E1 4.3524,E2 476.0096} C_DIS
LIN {X 124.3165,Y -60.2339,Z 183,A -21.7769,B 4.2007,C 0.2705,E1 4.3542,E2 474.5443} C_DIS
LIN {X 125.746,Y -57.1914,Z 183,A -20.449,B 4.2009,C 0.2677,E1 4.3558,E2 473.224} C_DIS
LIN {X 127.1367,Y -54.0293,Z 183,A -18.9353,B 4.2012,C 0.2629,E1 4.3575,E2 471.6985} C_DIS
LIN {X 128.6465,Y -50.3222,Z 183,A -17.63,B 4.2012,C 0.2629,E1 4.3588,E2 470.4382} C_DIS
LIN {X 129.6612,Y -47.6536,Z 183,A -16.3086,B 4.2015,C 0.258,E1 4.3601,E2 469.098} C_DIS
LIN {X 130.7952,Y -44.4466,Z 183,A -14.944,B 4.2017,C 0.2548,E1 4.3613,E2 467.7383} C_DIS
LIN {X 131.8442,Y -41.2312,Z 183,A -13.4704,B 4.202,C 0.2501,E1 4.3626,E2 466.2543} C_DIS
LIN {X 132.8575,Y -37.8353,Z 183,A -12.0719,B 4.2022,C 0.247,E1 4.3637,E2 464.8639} C_DIS
LIN {X 133.8399,Y -34.1926,Z 183,A -10.8706,B 4.2022,C 0.2472,E1 4.3645,E2 463.7087} C_DIS
LIN {X 134.5921,Y -31.1014,Z 183,A -9.3482,B 4.2025,C 0.241,E1 4.3655,E2 462.1589} C_DIS
LIN {X 135.3217,Y -27.7544,Z 183,A -8.0065,B 4.2027,C 0.2381,E1 4.3663,E2 460.8263} C_DIS
LIN {X 135.9587,Y -24.4435,Z 183,A -6.64,B 4.2029,C 0.2346,E1 4.367,E2 459.4629} C_DIS
LIN {X 136.6355,Y -20.3382,Z 183,A -4.9885,B 4.2031,C 0.2307,E1 4.3677,E2 457.8199} C_DIS
LIN {X 137.1413,Y -16.57,Z 183,A -3.674,B 4.2031,C 0.2295,E1 4.3681,E2 456.5381} C_DIS
LIN {X 137.4307,Y -13.9891,Z 183,A -2.2755,B 4.2035,C 0.2224,E1 4.3686,E2 455.0972} C_DIS
LIN {X 137.7571,Y -10.2624,Z 183,A -0.9021,B 4.2036,C 0.2203,E1 4.3689,E2 453.7457} C_DIS
LIN {X 137.9709,Y -6.8076,Z 183,A 0.4675,B 4.2038,C 0.2171,E1 4.3691,E2 452.3837} C_DIS
LIN {X 138.1068,Y -3.0662,Z 183,A 1.9564,B 4.204,C 0.2135,E1 4.3691,E2 450.902} C_DIS
LIN {X 138.1419,Y 0.1091,Z 183,A 3.3853,B 4.2043,C 0.2083,E1 4.3692,E2 449.4577} C_DIS
LIN {X 138.091,Y 3.6361,Z 183,A 4.6745,B 4.2043,C 0.2064,E1 4.3692,E2 448.1899} C_DIS
LIN {X 137.9253,Y 7.7136,Z 183,A 6.2864,B 4.2045,C 0.2026,E1 4.3689,E2 446.5873} C_DIS
LIN {X 137.7148,Y 10.841,Z 183,A 7.6977,B 4.2048,C 0.1975,E1 4.3686,E2 445.1608} C_DIS
LIN {X 137.3679,Y 14.5731,Z 183,A 8.9997,B 4.2048,C 0.1963,E1 4.3683,E2 443.8902} C_DIS
LIN {X 136.9945,Y 17.7428,Z 183,A 10.3509,B 4.205,C 0.1923,E1 4.3678,E2 442.5347} C_DIS
LIN {X 136.3883,Y 21.9347,Z 183,A 12.0378,B 4.2052,C 0.1882,E1 4.3671,E2 440.8558} C_DIS
LIN {X 135.8347,Y 25.1365,Z 183,A 13.3437,B 4.2053,C 0.185,E1 4.3665,E2 439.5544} C_DIS
LIN {X 135.201,Y 28.3479,Z 183,A 14.6597,B 4.2055,C 0.1817,E1 4.3657,E2 438.243} C_DIS
LIN {X 134.4023,Y 31.9134,Z 183,A 16.1724,B 4.2057,C 0.1776,E1 4.3648,E2 436.7296} C_DIS
LIN {X 133.5373,Y 35.3562,Z 183,A 17.3471,B 4.2057,C 0.1772,E1 4.364,E2 435.5921} C_DIS
LIN {X 132.8085,Y 38.0106,Z 183,A 18.6632,B 4.2059,C 0.172,E1 4.363,E2 434.2533} C_DIS
LIN {X 131.7359,Y 41.5702,Z 183,A 20.1764,B 4.206,C 0.1681,E1 4.3617,E2 432.7428} C_DIS
LIN {X 130.631,Y 44.9204,Z 183,A 21.399,B 4.206,C 0.1672,E1 4.3607,E2 431.5501} C_DIS
LIN {X 129.6612,Y 47.6536,Z 183,A 22.7446,B 4.2063,C 0.1622,E1 4.3594,E2 430.1859} C_DIS
LIN {X 128.4418,Y 50.8489,Z 183,A 24.1207,B 4.2064,C 0.159,E1 4.358,E2 428.8145} C_DIS
LIN {X 126.9483,Y 54.4651,Z 183,A 25.6116,B 4.2065,C 0.1564,E1 4.3564,E2 427.3395} C_DIS
LIN {X 125.746,Y 57.1914,Z 183,A 26.8954,B 4.2066,C 0.1526,E1 4.3549,E2 426.0491} C_DIS
LIN {X 124.2697,Y 60.3319,Z 183,A 28.2929,B 4.2068,C 0.1494,E1 4.3533,E2 424.6563} C_DIS
LIN {X 122.5076,Y 63.8297,Z 183,A 29.9032,B 4.2068,C 0.1454,E1 4.3512,E2 423.047} C_DIS
LIN {X 120.3664,Y 67.7838,Z 183,A 31.7254,B 4.207,C 0.1413,E1 4.3488,E2 421.2296} C_DIS
LIN {X 118.2674,Y 71.3831,Z 183,A 33.4493,B 4.2072,C 0.1371,E1 4.3463,E2 419.5056} C_DIS
LIN {X 115.8012,Y 75.3181,Z 183,A 35.2787,B 4.2072,C 0.1337,E1 4.3436,E2 417.6879} C_DIS
LIN {X 113.3274,Y 78.9913,Z 183,A 37.066,B 4.2074,C 0.1299,E1 4.3408,E2 415.9062} C_DIS
LIN {X 110.7216,Y 82.6042,Z 183,A 38.8624,B 4.2075,C 0.1263,E1 4.3378,E2 414.1157} C_DIS
LIN {X 108.0108,Y 86.1184,Z 183,A 40.6574,B 4.2076,C 0.1227,E1 4.3347,E2 412.326} C_DIS
LIN {X 105.1747,Y 89.5601,Z 183,A 42.487,B 4.2077,C 0.1189,E1 4.3314,E2 410.4985} C_DIS
LIN {X 102.225,Y 92.9126,Z 183,A 44.2661,B 4.2078,C 0.1158,E1 4.3281,E2 408.7282} C_DIS
LIN {X 99.1662,Y 96.1706,Z 183,A 46.0855,B 4.2079,C 0.1123,E1 4.3246,E2 406.9127} C_DIS
LIN {X 96.1706,Y 99.1662,Z 183,A 47.8332,B 4.2079,C 0.1089,E1 4.3212,E2 405.1659} C_DIS
LIN {X 92.9126,Y 102.225,Z 183,A 49.6439,B 4.2081,C 0.1057,E1 4.3175,E2 403.3604} C_DIS
LIN {X 89.4042,Y 105.3072,Z 183,A 51.4986,B 4.2081,C 0.103,E1 4.3136,E2 401.5158} C_DIS
LIN {X 85.9449,Y 108.1489,Z 183,A 53.3119,B 4.2082,C 0.1001,E1 4.3096,E2 399.7077} C_DIS
LIN {X 82.4979,Y 110.8007,Z 183,A 55.0958,B 4.2082,C 0.0972,E1 4.3057,E2 397.9261} C_DIS
LIN {X 78.9913,Y 113.3274,Z 183,A 56.875,B 4.2083,C 0.0943,E1 4.3016,E2 396.1486} C_DIS
LIN {X 75.3181,Y 115.8012,Z 183,A 58.6756,B 4.2084,C 0.0918,E1 4.2974,E2 394.3524} C_DIS
LIN {X 71.3831,Y 118.2674,Z 183,A 60.5221,B 4.2084,C 0.0897,E1 4.2931,E2 392.516} C_DIS
LIN {X 67.5614,Y 120.4914,Z 183,A 62.3186,B 4.2084,C 0.0874,E1 4.2887,E2 390.7242} C_DIS
LIN {X 63.8763,Y 122.4831,Z 183,A 64.0252,B 4.2085,C 0.0853,E1 4.2845,E2 389.0216} C_DIS
LIN {X 60.3319,Y 124.2697,Z 183,A 65.6066,B 4.2085,C 0.0839,E1 4.2806,E2 387.4484} C_DIS
LIN {X 57.1914,Y 125.746,Z 183,A 67.1507,B 4.2086,C 0.081,E1 4.2766,E2 385.8914} C_DIS
LIN {X 54.0293,Y 127.1367,Z 183,A 68.4342,B 4.2086,C 0.0808,E1 4.2734,E2 384.6267} C_DIS
LIN {X 50.8489,Y 128.4418,Z 183,A 69.8396,B 4.2086,C 0.0795,E1 4.2697,E2 383.224} C_DIS
LIN {X 47.1743,Y 129.834,Z 183,A 71.4431,B 4.2086,C 0.078,E1 4.2655,E2 381.624} C_DIS
LIN {X 44.4466,Y 130.7952,Z 183,A 72.6309,B 4.2087,C 0.077,E1 4.2624,E2 380.438} C_DIS
LIN {X 41.2312,Y 131.8442,Z 183,A 74.0165,B 4.2087,C 0.0758,E1 4.2587,E2 379.0548} C_DIS
LIN {X 38.0106,Y 132.8085,Z 183,A 75.5278,B 4.2087,C 0.0735,E1 4.2546,E2 377.5293} C_DIS
LIN {X 34.1926,Y 133.8399,Z 183,A 76.8559,B 4.2087,C 0.0753,E1 4.2512,E2 376.2402} C_DIS
LIN {X 31.5659,Y 134.486,Z 183,A 78.1274,B 4.2087,C 0.073,E1 4.2476,E2 374.9505} C_DIS
LIN {X 28.3479,Y 135.201,Z 183,A 79.4818,B 4.2087,C 0.0722,E1 4.244,E2 373.5982} C_DIS
LIN {X 25.1365,Y 135.8347,Z 183,A 80.9532,B 4.2088,C 0.0703,E1 4.2399,E2 372.113} C_DIS
LIN {X 21.3357,Y 136.4811,Z 183,A 82.1919,B 4.2088,C 0.0729,E1 4.2366,E2 370.9194} C_DIS
LIN {X 18.7451,Y 136.8632,Z 183,A 83.6495,B 4.2088,C 0.0688,E1 4.2324,E2 369.4162} C_DIS
LIN {X 15.5702,Y 137.2606,Z 183,A 84.8103,B 4.2088,C 0.0699,E1 4.2293,E2 368.2765} C_DIS
LIN {X 11.832,Y 137.6311,Z 183,A 86.39,B 4.2088,C 0.0691,E1 4.2249,E2 366.6947} C_DIS
LIN {X 7.7136,Y 137.9253,Z 183,A 88.063,B 4.2088,C 0.0691,E1 4.2202,E2 365.0273} C_DIS
LIN {X 4.6091,Y 138.064,Z 183,A 89.3468,B 4.2088,C 0.0689,E1 4.2166,E2 363.7446} C_DIS
LIN {X 0.9647,Y 138.1355,Z 183,A 90.6457,B 4.2088,C 0.0707,E1 4.2131,E2 362.4726} C_DIS
LIN {X -2.0972,Y 138.123,Z 183,A 92.1776,B 4.2088,C 0.0682,E1 4.2087,E2 360.909} C_DIS
LIN {X -5.1814,Y 138.0416,Z 183,A 93.4082,B 4.2088,C 0.0687,E1 4.2053,E2 359.685} C_DIS
LIN {X -9.2745,Y 137.8292,Z 183,A 95.1127,B 4.2088,C 0.0688,E1 4.2005,E2 357.9808} C_DIS
LIN {X -12.9949,Y 137.5262,Z 183,A 96.6677,B 4.2088,C 0.069,E1 4.1962,E2 356.4257} C_DIS
LIN {X -17.1556,Y 137.0715,Z 183,A 98.5594,B 4.2088,C 0.0681,E1 4.1909,E2 354.5157} C_DIS
LIN {X -21.9347,Y 136.3883,Z 183,A 100.4259,B 4.2088,C 0.07,E1 4.1858,E2 352.667} C_DIS
LIN {X -25.1365,Y 135.8347,Z 183,A 101.7828,B 4.2088,C 0.0705,E1 4.1821,E2 351.3098} C_DIS
LIN {X -28.3479,Y 135.201,Z 183,A 103.1509,B 4.2088,C 0.071,E1 4.1783,E2 349.9411} C_DIS
LIN {X -31.9385,Y 134.3962,Z 183,A 104.7103,B 4.2088,C 0.0716,E1 4.1741,E2 348.3784} C_DIS
LIN {X -35.3877,Y 133.5289,Z 183,A 105.9475,B 4.2088,C 0.0746,E1 4.1708,E2 347.1714} C_DIS
LIN {X -38.1813,Y 132.7585,Z 183,A 107.3267,B 4.2088,C 0.0739,E1 4.167,E2 345.7711} C_DIS
LIN {X -41.2312,Y 131.8442,Z 183,A 108.8635,B 4.2088,C 0.0731,E1 4.1629,E2 344.2085} C_DIS
LIN {X -44.9777,Y 130.6111,Z 183,A 110.1723,B 4.2087,C 0.0772,E1 4.1595,E2 342.941} C_DIS
LIN {X -47.6536,Y 129.6612,Z 183,A 111.5752,B 4.2087,C 0.0764,E1 4.1557,E2 341.5113} C_DIS
LIN {X -50.8489,Y 128.4418,Z 183,A 113.0119,B 4.2087,C 0.0776,E1 4.152,E2 340.0731} C_DIS
LIN {X -54.0293,Y 127.1367,Z 183,A 114.4575,B 4.2087,C 0.079,E1 4.1483,E2 338.6261} C_DIS
LIN {X -57.3244,Y 125.6844,Z 183,A 115.992,B 4.2087,C 0.0803,E1 4.1443,E2 337.0875} C_DIS
LIN {X -60.3319,Y 124.2697,Z 183,A 117.3725,B 4.2087,C 0.0819,E1 4.1409,E2 335.7078} C_DIS
LIN {X -63.4474,Y 122.7083,Z 183,A 118.9179,B 4.2086,C 0.0829,E1 4.137,E2 334.151} C_DIS
LIN {X -67.3014,Y 120.6375,Z 183,A 120.8076,B 4.2086,C 0.0847,E1 4.1323,E2 332.2533} C_DIS
LIN {X -71.1046,Y 118.4358,Z 183,A 122.6193,B 4.2085,C 0.0873,E1 4.128,E2 330.4443} C_DIS
LIN {X -74.8504,Y 116.1048,Z 183,A 124.4839,B 4.2085,C 0.0897,E1 4.1236,E2 328.5767} C_DIS
LIN {X -78.5322,Y 113.6468,Z 183,A 126.3989,B 4.2084,C 0.0919,E1 4.1191,E2 326.6532} C_DIS
LIN {X -82.1981,Y 111.024,Z 183,A 128.2473,B 4.2084,C 0.0951,E1 4.115,E2 324.8089} C_DIS
LIN {X -85.6787,Y 108.3608,Z 183,A 130.1215,B 4.2083,C 0.0978,E1 4.1108,E2 322.9291} C_DIS
LIN {X -89.1312,Y 105.5392,Z 183,A 132.0408,B 4.2083,C 0.1006,E1 4.1067,E2 321.0025} C_DIS
LIN {X -92.4953,Y 102.6037,Z 183,A 133.907,B 4.2081,C 0.1039,E1 4.1028,E2 319.136} C_DIS
LIN {X -95.7655,Y 99.5583,Z 183,A 135.8474,B 4.2081,C 0.1068,E1 4.0988,E2 317.1862} C_DIS
LIN {X -98.9484,Y 96.3956,Z 183,A 137.7501,B 4.208,C 0.1102,E1 4.0951,E2 315.2799} C_DIS
LIN {X -102.06,Y 93.0946,Z 183,A 139.6627,B 4.2079,C 0.1139,E1 4.0915,E2 313.3649} C_DIS
LIN {X -104.9611,Y 89.8113,Z 183,A 141.5484,B 4.2078,C 0.1172,E1 4.088,E2 311.4721} C_DIS
LIN {X -107.8058,Y 86.376,Z 183,A 143.4478,B 4.2077,C 0.1209,E1 4.0846,E2 309.568} C_DIS
LIN {X -110.5333,Y 82.857,Z 183,A 145.3025,B 4.2075,C 0.125,E1 4.0815,E2 307.7138} C_DIS
LIN {X -113.1402,Y 79.2603,Z 183,A 147.2389,B 4.2075,C 0.1286,E1 4.0783,E2 305.7671} C_DIS
LIN {X -115.6233,Y 75.592,Z 183,A 149.0863,B 4.2073,C 0.1328,E1 4.0755,E2 303.9199} C_DIS
LIN {X -117.9876,Y 71.8458,Z 183,A 151.0224,B 4.2072,C 0.1366,E1 4.0726,E2 301.973} C_DIS
LIN {X -120.2076,Y 68.0664,Z 183,A 152.8493,B 4.207,C 0.141,E1 4.0701,E2 300.1465} C_DIS
LIN {X -121.8958,Y 64.9947,Z 183,A 154.2691,B 4.207,C 0.1448,E1 4.0682,E2 298.7322} C_DIS
LIN {X -123.6549,Y 61.5783,Z 183,A 155.778,B 4.2068,C 0.1494,E1 4.0663,E2 297.2351} C_DIS
LIN {X -125.0185,Y 58.7645,Z 183,A 157.2487,B 4.2067,C 0.1515,E1 4.0645,E2 295.7437} C_DIS
LIN {X -126.452,Y 55.6128,Z 183,A 158.7299,B 4.2066,C 0.155,E1 4.0628,E2 294.258} C_DIS
LIN {X -127.7999,Y 52.4412,Z 183,A 160.2045,B 4.2064,C 0.1584,E1 4.0612,E2 292.7789} C_DIS
LIN {X -129.1648,Y 48.979,Z 183,A 161.6856,B 4.2063,C 0.1629,E1 4.0597,E2 291.3069} C_DIS
LIN {X -130.2389,Y 46.0514,Z 183,A 163.1324,B 4.2062,C 0.1654,E1 4.0584,E2 289.8419} C_DIS
LIN {X -131.3303,Y 42.8398,Z 183,A 164.6641,B 4.206,C 0.1683,E1 4.057,E2 288.2955} C_DIS
LIN {X -132.3369,Y 39.6214,Z 183,A 166.029,B 4.2059,C 0.1723,E1 4.0559,E2 286.936} C_DIS
LIN {X -133.3957,Y 35.8871,Z 183,A 167.7126,B 4.2057,C 0.1763,E1 4.0546,E2 285.2442} C_DIS
LIN {X -134.1331,Y 33.0299,Z 183,A 168.8986,B 4.2056,C 0.1799,E1 4.0538,E2 284.064} C_DIS
LIN {X -134.8537,Y 29.9562,Z 183,A 170.3091,B 4.2054,C 0.1829,E1 4.0529,E2 282.6418} C_DIS
LIN {X -135.5279,Y 26.7412,Z 183,A 171.7171,B 4.2053,C 0.1864,E1 4.0522,E2 281.2291} C_DIS
LIN {X -136.2127,Y 22.9872,Z 183,A 173.3109,B 4.2051,C 0.1907,E1 4.0514,E2 279.635} C_DIS
LIN {X -136.6355,Y 20.3382,Z 183,A 174.5023,B 4.205,C 0.1933,E1 4.0509,E2 278.4345} C_DIS
LIN {X -137.1413,Y 16.57,Z 183,A 175.9073,B 4.2047,C 0.1988,E1 4.0504,E2 277.0525} C_DIS
LIN {X -137.4307,Y 13.9891,Z 183,A 177.4082,B 4.2047,C 0.1992,E1 4.0499,E2 275.4986} C_DIS
LIN {X -137.7661,Y 10.1389,Z 183,A 178.8736,B 4.2044,C 0.2046,E1 4.0496,E2 274.0519} C_DIS
LIN {X -138.0035,Y 6.1584,Z 183,A -179.3881,B 4.2042,C 0.2088,E1 4.0493,E2 272.3041} C_DIS
LIN {X -138.1068,Y 3.0662,Z 183,A -178.0617,B 4.2041,C 0.2122,E1 4.0493,E2 270.9731} C_DIS
LIN {X -138.1419,Y -0.1091,Z 183,A -176.53,B 4.2039,C 0.2145,E1 4.0493,E2 269.4149} C_DIS
LIN {X -138.0837,Y -3.898,Z 183,A -175.0846,B 4.2037,C 0.2198,E1 4.0493,E2 267.9866} C_DIS
LIN {X -137.9253,Y -7.7136,Z 183,A -173.4248,B 4.2035,C 0.2238,E1 4.0495,E2 266.3183} C_DIS
LIN {X -137.6646,Y -11.4356,Z 183,A -171.8221,B 4.2032,C 0.2278,E1 4.0499,E2 264.7095} C_DIS
LIN {X -137.3679,Y -14.5731,Z 183,A -170.4511,B 4.2031,C 0.2311,E1 4.0503,E2 263.3312} C_DIS
LIN {X -136.9945,Y -17.7428,Z 183,A -169.0899,B 4.2029,C 0.2345,E1 4.0507,E2 261.966} C_DIS
LIN {X -136.3883,Y -21.9347,Z 183,A -167.2689,B 4.2026,C 0.239,E1 4.0515,E2 260.138} C_DIS
LIN {X -135.8347,Y -25.1365,Z 183,A -165.7427,B 4.2025,C 0.2417,E1 4.0523,E2 258.5896} C_DIS
LIN {X -135.1144,Y -28.7487,Z 183,A -164.2984,B 4.2022,C 0.2464,E1 4.0531,E2 257.1569} C_DIS
LIN {X -134.3426,Y -32.1608,Z 183,A -163.0192,B 4.2019,C 0.2515,E1 4.0539,E2 255.9007} C_DIS
LIN {X -133.6889,Y -34.7878,Z 183,A -161.4934,B 4.2019,C 0.252,E1 4.0549,E2 254.3236} C_DIS
LIN {X -132.7032,Y -38.3704,Z 183,A -160.0161,B 4.2016,C 0.2565,E1 4.0561,E2 252.8553} C_DIS
LIN {X -131.8442,Y -41.2312,Z 183,A -158.7441,B 4.2014,C 0.2597,E1 4.0571,E2 251.5798} C_DIS
LIN {X -130.7952,Y -44.4466,Z 183,A -157.2927,B 4.2012,C 0.2631,E1 4.0584,E2 250.1229} C_DIS
LIN {X -129.5535,Y -47.9412,Z 183,A -155.8185,B 4.2009,C 0.2676,E1 4.0598,E2 248.6577} C_DIS
LIN {X -128.4418,Y -50.8489,Z 183,A -154.2417,B 4.2009,C 0.269,E1 4.0614,E2 247.0446} C_DIS
LIN {X -127.0621,Y -54.2018,Z 183,A -152.8842,B 4.2005,C 0.2739,E1 4.0629,E2 245.7067} C_DIS
LIN {X -125.746,Y -57.1914,Z 183,A -151.413,B 4.2003,C 0.2766,E1 4.0646,E2 244.2211} C_DIS
LIN {X -124.0967,Y -60.6827,Z 183,A -149.9083,B 4.2,C 0.2813,E1 4.0664,E2 242.7296} C_DIS
LIN {X -122.7083,Y -63.4474,Z 183,A -148.3577,B 4.2,C 0.2826,E1 4.0684,E2 241.1449} C_DIS
LIN {X -120.6375,Y -67.3014,Z 183,A -146.4438,B 4.1997,C 0.2864,E1 4.071,E2 239.2188} C_DIS
LIN {X -118.4108,Y -71.1459,Z 183,A -144.5693,B 4.1994,C 0.2906,E1 4.0736,E2 237.3408} C_DIS
LIN {X -116.1048,Y -74.8504,Z 183,A -142.7221,B 4.1991,C 0.2945,E1 4.0764,E2 235.4894} C_DIS
LIN {X -113.6468,Y -78.5322,Z 183,A -140.7901,B 4.1989,C 0.2981,E1 4.0795,E2 233.5454} C_DIS
LIN {X -111.0645,Y -82.1437,Z 183,A -138.8957,B 4.1986,C 0.3018,E1 4.0826,E2 231.6446} C_DIS
LIN {X -108.3608,Y -85.6787,Z 183,A -137.0421,B 4.1983,C 0.3058,E1 4.0858,E2 229.7905} C_DIS
LIN {X -105.5392,Y -89.1312,Z 183,A -135.1435,B 4.198,C 0.3093,E1 4.0892,E2 227.8858} C_DIS
LIN {X -102.6037,Y -92.4953,Z 183,A -133.2441,B 4.1978,C 0.3127,E1 4.0927,E2 225.9807} C_DIS
LIN {X -99.5583,Y -95.7655,Z 183,A -131.3025,B 4.1976,C 0.3157,E1 4.0964,E2 224.0279} C_DIS
LIN {X -96.4078,Y -98.9365,Z 183,A -129.4046,B 4.1973,C 0.319,E1 4.1002,E2 222.1245} C_DIS
LIN {X -93.1571,Y -102.0033,Z 183,A -127.509,B 4.1971,C 0.3221,E1 4.1041,E2 220.2236} C_DIS
LIN {X -89.8113,Y -104.9611,Z 183,A -125.6168,B 4.1969,C 0.325,E1 4.1081,E2 218.3264} C_DIS
LIN {X -86.376,Y -107.8058,Z 183,A -123.7289,B 4.1966,C 0.3279,E1 4.1122,E2 216.4336} C_DIS
LIN {X -82.857,Y -110.5333,Z 183,A -121.8882,B 4.1964,C 0.3309,E1 4.1163,E2 214.5938} C_DIS
LIN {X -79.2603,Y -113.1402,Z 183,A -119.9692,B 4.1962,C 0.3331,E1 4.1207,E2 212.6648} C_DIS
LIN {X -75.5337,Y -115.6611,Z 183,A -118.131,B 4.196,C 0.3361,E1 4.125,E2 210.8303} C_DIS
LIN {X -71.8586,Y -117.9799,Z 183,A -116.2818,B 4.1958,C 0.3382,E1 4.1294,E2 208.9748} C_DIS
LIN {X -68.0664,Y -120.2076,Z 183,A -114.3936,B 4.1957,C 0.34,E1 4.134,E2 207.0781} C_DIS
LIN {X -64.9947,Y -121.8958,Z 183,A -113.0316,B 4.1955,C 0.3426,E1 4.1373,E2 205.7281} C_DIS
LIN {X -61.8929,Y -123.4997,Z 183,A -111.5639,B 4.1953,C 0.3441,E1 4.141,E2 204.2577} C_DIS
LIN {X -58.4539,Y -125.1622,Z 183,A -109.9466,B 4.1953,C 0.3456,E1 4.1451,E2 202.6358} C_DIS
LIN {X -55.6128,Y -126.452,Z 183,A -108.6506,B 4.1951,C 0.3469,E1 4.1484,E2 201.3394} C_DIS
LIN {X -52.4412,Y -127.7999,Z 183,A -107.1202,B 4.1951,C 0.3474,E1 4.1523,E2 199.7954} C_DIS
LIN {X -49.0179,Y -129.1502,Z 183,A -105.7577,B 4.1948,C 0.3502,E1 4.1558,E2 198.4543} C_DIS
LIN {X -46.0514,Y -130.2389,Z 183,A -104.3422,B 4.1948,C 0.3504,E1 4.1596,E2 197.0247} C_DIS
LIN {X -42.6865,Y -131.3793,Z 183,A -102.9163,B 4.1947,C 0.3519,E1 4.1634,E2 195.6048} C_DIS
LIN {X -39.4639,Y -132.383,Z 183,A -101.3453,B 4.1947,C 0.3513,E1 4.1676,E2 194.0106} C_DIS
LIN {X -35.804,Y -133.4179,Z 183,A -99.8602,B 4.1946,C 0.3532,E1 4.1716,E2 192.5375} C_DIS
LIN {X -31.5659,Y -134.486,Z 183,A -98.0377,B 4.1946,C 0.354,E1 4.1765,E2 190.7132} C_DIS
LIN {X -28.3479,Y -135.201,Z 183,A -96.5111,B 4.1946,C 0.3532,E1 4.1808,E2 189.165} C_DIS
LIN {X -25.1365,Y -135.8347,Z 183,A -95.2227,B 4.1945,C 0.3544,E1 4.1843,E2 187.8853} C_DIS
LIN {X -21.9347,Y -136.3883,Z 183,A -93.9519,B 4.1944,C 0.3555,E1 4.1878,E2 186.6244} C_DIS
LIN {X -18.7451,Y -136.8632,Z 183,A -92.4547,B 4.1944,C 0.3544,E1 4.192,E2 185.1053} C_DIS
LIN {X -15.0821,Y -137.3131,Z 183,A -91.0508,B 4.1944,C 0.3559,E1 4.1958,E2 183.7177} C_DIS
LIN {X -11.6703,Y -137.6448,Z 183,A -89.6955,B 4.1943,C 0.3567,E1 4.1996,E2 182.3707} C_DIS
LIN {X -7.7136,Y -137.9253,Z 183,A -88.0169,B 4.1943,C 0.3564,E1 4.2043,E2 180.687} C_DIS
LIN {X -4.6091,Y -138.064,Z 183,A -86.7306,B 4.1943,C 0.3564,E1 4.2079,E2 179.4005} C_DIS
LIN {X -0.9647,Y -138.1355,Z 183,A -85.186,B 4.1943,C 0.3559,E1 4.2122,E2 177.8507} C_DIS
LIN {X -0.9647,Y -138.1355,Z 183,A -85.186,B 4.1943,C 0.3559,E1 4.2122,E2 177.8507} C_DIS
Enddeposition()
LIN {X 0.976,Y -139.0352,Z 183,A -84.4003,B 4.1502,C 0.3571,E1 4.1703,E2 177.111} C_DIS
Startdeposition()
$VEL.CP = VEL_PRINT
LIN {X -3.4633,Y -138.9972,Z 183,A -86.7707,B 4.1497,C 0.3626,E1 4.1635,E2 179.5547} C_DIS
LIN {X -7.0011,Y -138.8633,Z 183,A -88.3181,B 4.1497,C 0.3635,E1 4.1591,E2 181.1146} C_DIS
LIN {X -11.5646,Y -138.5579,Z 183,A -90.1366,B 4.1497,C 0.3627,E1 4.1541,E2 182.925} C_DIS
LIN {X -15.0984,Y -138.2176,Z 183,A -91.6264,B 4.1497,C 0.3627,E1 4.1499,E2 184.419} C_DIS
LIN {X -19.3028,Y -137.6936,Z 183,A -93.3827,B 4.1497,C 0.3625,E1 4.1451,E2 186.1773} C_DIS
LIN {X -23.232,Y -137.0853,Z 183,A -95.3152,B 4.1495,C 0.3646,E1 4.1396,E2 188.1494} C_DIS
LIN {X -26.7734,Y -136.4391,Z 183,A -96.4432,B 4.1499,C 0.3608,E1 4.1367,E2 189.2308} C_DIS
LIN {X -34.2711,Y -134.7496,Z 183,A -99.7898,B 4.1499,C 0.3608,E1 4.1275,E2 192.6022} C_DIS
LIN {X -38.7714,Y -133.5246,Z 183,A -101.5725,B 4.1501,C 0.3584,E1 4.1227,E2 194.367} C_DIS
LIN {X -42.2948,Y -132.4503,Z 183,A -103.1369,B 4.1501,C 0.3577,E1 4.1185,E2 195.9378} C_DIS
LIN {X -45.4342,Y -131.4065,Z 183,A -104.7763,B 4.1501,C 0.3591,E1 4.1141,E2 197.6141} C_DIS
LIN {X -50.1301,Y -129.6879,Z 183,A -106.5924,B 4.1504,C 0.3552,E1 4.1094,E2 199.3983} C_DIS
LIN {X -53.3262,Y -128.4068,Z 183,A -107.9937,B 4.1504,C 0.3537,E1 4.1058,E2 200.7974} C_DIS
LIN {X -56.3286,Y -127.1189,Z 183,A -109.5756,B 4.1504,C 0.3543,E1 4.1017,E2 202.4107} C_DIS
LIN {X -66.2602,Y -122.2382,Z 183,A -114.1492,B 4.1509,C 0.3492,E1 4.0903,E2 206.9866} C_DIS
LIN {X -70.3309,Y -119.9418,Z 183,A -116.0682,B 4.1511,C 0.3466,E1 4.0856,E2 208.9048} C_DIS
LIN {X -74.6968,Y -117.2729,Z 183,A -118.3216,B 4.1512,C 0.3448,E1 4.0802,E2 211.1773} C_DIS
LIN {X -78.346,Y -114.8674,Z 183,A -120.9736,B 4.1509,C 0.3488,E1 4.0739,E2 213.9405} C_DIS
LIN {X -84.1869,Y -110.6577,Z 183,A -123.1053,B 4.1518,C 0.3376,E1 4.0694,E2 215.9632} C_DIS
LIN {X -87.7747,Y -107.8338,Z 183,A -125.0234,B 4.1521,C 0.3348,E1 4.0652,E2 217.8858} C_DIS
LIN {X -91.2985,Y -104.8669,Z 183,A -126.9492,B 4.1523,C 0.3317,E1 4.0611,E2 219.815} C_DIS
LIN {X -94.7071,Y -101.7989,Z 183,A -128.8485,B 4.1526,C 0.3283,E1 4.0571,E2 221.7153} C_DIS
LIN {X -97.8492,Y -98.7828,Z 183,A -130.7087,B 4.1528,C 0.3254,E1 4.0534,E2 223.5838} C_DIS
LIN {X -100.9771,Y -95.5831,Z 183,A -132.6115,B 4.153,C 0.3222,E1 4.0497,E2 225.494} C_DIS
LIN {X -104.0551,Y -92.2226,Z 183,A -134.5247,B 4.1533,C 0.3186,E1 4.0461,E2 227.4114} C_DIS
LIN {X -107.0053,Y -88.7825,Z 183,A -136.4241,B 4.1536,C 0.3149,E1 4.0427,E2 229.3145} C_DIS
LIN {X -109.788,Y -85.3175,Z 183,A -138.3194,B 4.1539,C 0.3114,E1 4.0394,E2 231.2177} C_DIS
LIN {X -112.4325,Y -81.8012,Z 183,A -140.2021,B 4.1541,C 0.3079,E1 4.0362,E2 233.1089} C_DIS
LIN {X -115.053,Y -78.0723,Z 183,A -142.1231,B 4.1544,C 0.3039,E1 4.0332,E2 235.0348} C_DIS
LIN {X -117.4631,Y -74.3971,Z 183,A -144.0786,B 4.1547,C 0.3007,E1 4.0302,E2 237.0085} C_DIS
LIN {X -120.2202,Y -69.8542,Z 183,A -146.7892,B 4.1547,C 0.299,E1 4.0263,E2 239.7856} C_DIS
LIN {X -122.737,Y -65.3308,Z 183,A -148.3742,B 4.1554,C 0.2901,E1 4.0243,E2 241.2989} C_DIS
LIN {X -124.5109,Y -61.8798,Z 183,A -150.0174,B 4.1557,C 0.2864,E1 4.0222,E2 242.9471} C_DIS
LIN {X -125.9405,Y -58.9176,Z 183,A -151.4691,B 4.1559,C 0.2836,E1 4.0204,E2 244.4108} C_DIS
LIN {X -127.2043,Y -56.1378,Z 183,A -152.9669,B 4.1559,C 0.282,E1 4.0187,E2 245.939} C_DIS
LIN {X -129.2663,Y -51.2135,Z 183,A -155.0926,B 4.1564,C 0.2758,E1 4.0165,E2 248.0541} C_DIS
LIN {X -130.3437,Y -48.4003,Z 183,A -156.2669,B 4.1566,C 0.2721,E1 4.0153,E2 249.219} C_DIS
LIN {X -132.6464,Y -41.681,Z 183,A -159.3893,B 4.157,C 0.2656,E1 4.0126,E2 252.3651} C_DIS
LIN {X -133.8367,Y -37.6795,Z 183,A -161.0308,B 4.1574,C 0.2604,E1 4.0113,E2 253.9955} C_DIS
LIN {X -134.7062,Y -34.4422,Z 183,A -162.4679,B 4.1576,C 0.257,E1 4.0103,E2 255.439} C_DIS
LIN {X -135.5443,Y -30.9793,Z 183,A -163.9566,B 4.1578,C 0.2531,E1 4.0093,E2 256.9295} C_DIS
LIN {X -136.2238,Y -27.8401,Z 183,A -165.3861,B 4.158,C 0.2501,E1 4.0085,E2 258.3718} C_DIS
LIN {X -137.0406,Y -23.4999,Z 183,A -167.5202,B 4.1582,C 0.247,E1 4.0074,E2 260.545} C_DIS
LIN {X -137.8299,Y -18.3026,Z 183,A -169.4819,B 4.1586,C 0.2397,E1 4.0066,E2 262.4792} C_DIS
LIN {X -138.321,Y -14.1377,Z 183,A -171.5327,B 4.1588,C 0.2368,E1 4.006,E2 264.5702} C_DIS
LIN {X -138.7465,Y -9.0383,Z 183,A -173.9969,B 4.159,C 0.2331,E1 4.0055,E2 267.0781} C_DIS
LIN {X -138.969,Y -4.4761,Z 183,A -175.5361,B 4.1594,C 0.2257,E1 4.0054,E2 268.5724} C_DIS
LIN {X -139.0356,Y -1.2076,Z 183,A -177.1744,B 4.1595,C 0.2236,E1 4.0054,E2 270.2468} C_DIS
LIN {X -139.0198,Y 2.3584,Z 183,A -178.4275,B 4.1598,C 0.2181,E1 4.0054,E2 271.4714} C_DIS
LIN {X -138.7318,Y 9.277,Z 183,A 178.5966,B 4.1602,C 0.2108,E1 4.0058,E2 274.4609} C_DIS
LIN {X -138.4371,Y 12.9353,Z 183,A 177.0744,B 4.1604,C 0.2066,E1 4.0061,E2 275.9831} C_DIS
LIN {X -137.6307,Y 19.743,Z 183,A 174.0986,B 4.1607,C 0.1996,E1 4.0072,E2 278.9759} C_DIS
LIN {X -136.9126,Y 24.2282,Z 183,A 172.2155,B 4.161,C 0.1944,E1 4.0081,E2 280.859} C_DIS
LIN {X -136.1853,Y 28.029,Z 183,A 170.5428,B 4.1612,C 0.1905,E1 4.009,E2 282.5403} C_DIS
LIN {X -135.112,Y 32.8142,Z 183,A 168.5237,B 4.1614,C 0.1849,E1 4.0103,E2 284.5576} C_DIS
LIN {X -134.047,Y 36.9276,Z 183,A 166.7314,B 4.1616,C 0.1803,E1 4.0115,E2 286.3538} C_DIS
LIN {X -133.0785,Y 40.2769,Z 183,A 165.2143,B 4.1617,C 0.1769,E1 4.0127,E2 287.8798} C_DIS
LIN {X -132.0001,Y 43.6804,Z 183,A 163.7183,B 4.1619,C 0.1731,E1 4.014,E2 289.3778} C_DIS
LIN {X -130.8432,Y 47.0319,Z 183,A 162.2067,B 4.1621,C 0.1695,E1 4.0154,E2 290.8946} C_DIS
LIN {X -129.653,Y 50.2199,Z 183,A 160.7731,B 4.1621,C 0.166,E1 4.0169,E2 292.3309} C_DIS
LIN {X -128.3726,Y 53.4082,Z 183,A 159.2603,B 4.1623,C 0.1629,E1 4.0185,E2 293.8548} C_DIS
LIN {X -126.9895,Y 56.618,Z 183,A 157.804,B 4.1625,C 0.1593,E1 4.0201,E2 295.3119} C_DIS
LIN {X -125.3156,Y 60.233,Z 183,A 156.0731,B 4.1625,C 0.1557,E1 4.0222,E2 297.0527} C_DIS
LIN {X -123.4634,Y 63.9476,Z 183,A 154.2235,B 4.1627,C 0.1522,E1 4.0245,E2 298.9184} C_DIS
LIN {X -121.3026,Y 67.9571,Z 183,A 152.5736,B 4.1629,C 0.1461,E1 4.0267,E2 300.5383} C_DIS
LIN {X -119.0169,Y 71.8849,Z 183,A 150.3804,B 4.163,C 0.1437,E1 4.0299,E2 302.77} C_DIS
LIN {X -117.3491,Y 74.5777,Z 183,A 148.813,B 4.163,C 0.1422,E1 4.0323,E2 304.369} C_DIS
LIN {X -115.4855,Y 77.4315,Z 183,A 147.7275,B 4.1633,C 0.1369,E1 4.0339,E2 305.4137} C_DIS
LIN {X -111.7604,Y 82.7178,Z 183,A 144.8155,B 4.1633,C 0.1324,E1 4.0387,E2 308.3543} C_DIS
LIN {X -108.9603,Y 86.3723,Z 183,A 142.8796,B 4.1635,C 0.1285,E1 4.042,E2 310.2934} C_DIS
LIN {X -106.206,Y 89.7381,Z 183,A 141.0647,B 4.1636,C 0.1248,E1 4.0452,E2 312.1097} C_DIS
LIN {X -103.2647,Y 93.1077,Z 183,A 139.1399,B 4.1637,C 0.1215,E1 4.0488,E2 314.0431} C_DIS
LIN {X -100.1552,Y 96.4444,Z 183,A 137.2298,B 4.1638,C 0.1179,E1 4.0525,E2 315.9555} C_DIS
LIN {X -97.167,Y 99.454,Z 183,A 135.4522,B 4.1639,C 0.1146,E1 4.056,E2 317.7354} C_DIS
LIN {X -93.8781,Y 102.5643,Z 183,A 133.5411,B 4.164,C 0.1114,E1 4.0599,E2 319.6508} C_DIS
LIN {X -90.4688,Y 105.5839,Z 183,A 131.6067,B 4.164,C 0.1084,E1 4.064,E2 321.5908} C_DIS
LIN {X -86.9275,Y 108.5184,Z 183,A 129.6669,B 4.1642,C 0.1054,E1 4.0682,E2 323.5346} C_DIS
LIN {X -83.3444,Y 111.2938,Z 183,A 127.7418,B 4.1642,C 0.1027,E1 4.0725,E2 325.4654} C_DIS
LIN {X -79.6072,Y 113.9965,Z 183,A 125.8178,B 4.1643,C 0.0998,E1 4.0769,E2 327.3908} C_DIS
LIN {X -75.83,Y 116.5431,Z 183,A 123.9431,B 4.1643,C 0.097,E1 4.0813,E2 329.2639} C_DIS
LIN {X -72.2112,Y 118.8196,Z 183,A 122.1052,B 4.1644,C 0.095,E1 4.0857,E2 331.1099} C_DIS
LIN {X -68.2229,Y 121.1532,Z 183,A 120.1956,B 4.1644,C 0.0925,E1 4.0903,E2 333.0187} C_DIS
LIN {X -64.1418,Y 123.3614,Z 183,A 118.5457,B 4.1646,C 0.088,E1 4.0943,E2 334.6349} C_DIS
LIN {X -61.1334,Y 124.879,Z 183,A 116.9086,B 4.1646,C 0.0883,E1 4.0984,E2 336.3017} C_DIS
LIN {X -57.2776,Y 126.6944,Z 183,A 115.2399,B 4.1646,C 0.0856,E1 4.1026,E2 337.9584} C_DIS
LIN {X -53.9924,Y 128.1286,Z 183,A 113.6621,B 4.1646,C 0.0848,E1 4.1067,E2 339.5476} C_DIS
LIN {X -50.2099,Y 129.6569,Z 183,A 111.2811,B 4.1646,C 0.0887,E1 4.1131,E2 342.0131} C_DIS
LIN {X -45.1228,Y 131.5145,Z 183,A 109.5659,B 4.1646,C 0.0827,E1 4.1175,E2 343.6639} C_DIS
LIN {X -40.9113,Y 132.8844,Z 183,A 107.8931,B 4.1647,C 0.08,E1 4.1219,E2 345.3169} C_DIS
LIN {X -36.6022,Y 134.1375,Z 183,A 105.9379,B 4.1647,C 0.0796,E1 4.1272,E2 347.2841} C_DIS
LIN {X -33.0768,Y 135.0487,Z 183,A 104.5669,B 4.1647,C 0.0775,E1 4.1308,E2 348.6382} C_DIS
LIN {X -29.4157,Y 135.8922,Z 183,A 102.9103,B 4.1647,C 0.0776,E1 4.1354,E2 350.3072} C_DIS
LIN {X -25.9415,Y 136.5981,Z 183,A 101.5349,B 4.1648,C 0.0762,E1 4.1391,E2 351.6713} C_DIS
LIN {X -23.4132,Y 137.0551,Z 183,A 100.1279,B 4.1648,C 0.0787,E1 4.1431,E2 353.1206} C_DIS
LIN {X -18.2852,Y 137.8322,Z 183,A 98.2048,B 4.1648,C 0.0762,E1 4.1484,E2 355.0163} C_DIS
LIN {X -12.2106,Y 138.5034,Z 183,A 95.5855,B 4.1648,C 0.0765,E1 4.1557,E2 357.6467} C_DIS
LIN {X -5.3493,Y 138.9368,Z 183,A 92.8675,B 4.1648,C 0.0753,E1 4.1632,E2 360.3492} C_DIS
LIN {X -1.1344,Y 139.0356,Z 183,A 91.1161,B 4.1648,C 0.0754,E1 4.1681,E2 362.1016} C_DIS
LIN {X 2.6399,Y 139.0151,Z 183,A 89.5972,B 4.1648,C 0.0753,E1 4.1723,E2 363.6154} C_DIS
LIN {X 6.7861,Y 138.8741,Z 183,A 87.8793,B 4.1648,C 0.0757,E1 4.1771,E2 365.3336} C_DIS
LIN {X 10.2525,Y 138.6612,Z 183,A 86.4484,B 4.1648,C 0.0761,E1 4.1811,E2 366.7639} C_DIS
LIN {X 14.4651,Y 138.2857,Z 183,A 84.7058,B 4.1648,C 0.0767,E1 4.186,E2 368.5059} C_DIS
LIN {X 17.5959,Y 137.9225,Z 183,A 82.8207,B 4.1647,C 0.0828,E1 4.1914,E2 370.4624} C_DIS
LIN {X 22.5984,Y 137.1911,Z 183,A 81.3752,B 4.1647,C 0.0778,E1 4.1952,E2 371.829} C_DIS
LIN {X 31.5612,Y 135.4114,Z 183,A 77.5346,B 4.1647,C 0.0809,E1 4.2057,E2 375.678} C_DIS
LIN {X 35.4334,Y 134.4492,Z 183,A 76.0971,B 4.1647,C 0.0801,E1 4.2095,E2 377.0895} C_DIS
Enddeposition()
END
